	W =  90.000 deg,	P =   0.000 deg,	R =   90.000 deg
};
P[1529]{
   GP1:
	UF : 0, UT : 6,		CONFIG : 'N U T, 0, 0, 0',
	X =  489.358  mm,	Y =   -298.597  mm,	Z =   -262.804  mm,
	W =  90.000 deg,	P =   0.000 deg,	R =   90.000 deg
};
P[1530]{
   GP1:
	UF : 0, UT : 6,		CONFIG : 'N U T, 0, 0, 0',
	X =  488.486  mm,	Y =   -297.265  mm,	Z =   -263.052  mm,
	W =  90.000 deg,	P =   0.000 deg,	R =   90.000 deg
};
P[1531]{
   GP1:
	UF : 0, UT : 6,		CONFIG : 'N U T, 0, 0, 0',
	X =  487.911  mm,	Y =   -296.359  mm,	Z =   -263.179  mm,
	W =  90.000 deg,	P =   0.000 deg,	R =   90.000 deg
};
P[1532]{
   GP1:
	UF : 0, UT : 6,		CONFIG : 'N U T, 0, 0, 0',
	X =  487.436  mm,	Y =   -295.414  mm,	Z =   -263.006  mm,
	W =  90.000 deg,	P =   0.000 deg,	R =   90.000 deg
};
P[1533]{
   GP1:
	UF : 0, UT : 6,		CONFIG : 'N U T, 0, 0, 0',
	X =  485.822  mm,	Y =   -292.714  mm,	Z =   -263.142  mm,
	W =  90.000 deg,	P =   0.000 deg,	R =   90.000 deg
};
P[1534]{
   GP1:
	UF : 0, UT : 6,		CONFIG : 'N U T, 0, 0, 0',
	X =  485.360  mm,	Y =   -291.792  mm,	Z =   -262.970  mm,
	W =  90.000 deg,	P =   0.000 deg,	R =   90.000 deg
};
P[1535]{
   GP1:
	UF : 0, UT : 6,		CONFIG : 'N U T, 0, 0, 0',
	X =  484.532  mm,	Y =   -290.400  mm,	Z =   -263.029  mm,
	W =  90.000 deg,	P =   0.000 deg,	R =   90.000 deg
};
P[1536]{
   GP1:
	UF : 0, UT : 6,		CONFIG : 'N U T, 0, 0, 0',
	X =  483.396  mm,	Y =   -288.373  mm,	Z =   -262.945  mm,
	W =  90.000 deg,	P =   0.000 deg,	R =   90.000 deg
};
P[1537]{
   GP1:
	UF : 0, UT : 6,		CONFIG : 'N U T, 0, 0, 0',
	X =  482.953  mm,	Y =   -287.646  mm,	Z =   -263.001  mm,
	W =  90.000 deg,	P =   0.000 deg,	R =   90.000 deg
};
P[1538]{
   GP1:
	UF : 0, UT : 6,		CONFIG : 'N U T, 0, 0, 0',
	X =  482.093  mm,	Y =   -286.165  mm,	Z =   -263.010  mm,
	W =  90.000 deg,	P =   0.000 deg,	R =   90.000 deg
};
P[1539]{
   GP1:
	UF : 0, UT : 6,		CONFIG : 'N U T, 0, 0, 0',
	X =  480.613  mm,	Y =   -283.699  mm,	Z =   -263.148  mm,
	W =  90.000 deg,	P =   0.000 deg,	R =   90.000 deg
};
P[1540]{
   GP1:
	UF : 0, UT : 6,		CONFIG : 'N U T, 0, 0, 0',
	X =  479.567  mm,	Y =   -281.920  mm,	Z =   -263.196  mm,
	W =  90.000 deg,	P =   0.000 deg,	R =   90.000 deg
};
P[1541]{
   GP1:
	UF : 0, UT : 6,		CONFIG : 'N U T, 0, 0, 0',
	X =  478.631  mm,	Y =   -280.161  mm,	Z =   -263.002  mm,
	W =  90.000 deg,	P =   0.000 deg,	R =   90.000 deg
};
P[1542]{
   GP1:
	UF : 0, UT : 6,		CONFIG : 'N U T, 0, 0, 0',
	X =  478.100  mm,	Y =   -279.216  mm,	Z =   -262.965  mm,
	W =  90.000 deg,	P =   0.000 deg,	R =   90.000 deg
};
P[1543]{
   GP1:
	UF : 0, UT : 6,		CONFIG : 'N U T, 0, 0, 0',
	X =  477.160  mm,	Y =   -277.535  mm,	Z =   -262.892  mm,
	W =  90.000 deg,	P =   0.000 deg,	R =   90.000 deg
};
P[1544]{
   GP1:
	UF : 0, UT : 6,		CONFIG : 'N U T, 0, 0, 0',
	X =  476.282  mm,	Y =   -276.005  mm,	Z =   -262.880  mm,
	W =  90.000 deg,	P =   0.000 deg,	R =   90.000 deg
};
P[1545]{
   GP1:
	UF : 0, UT : 6,		CONFIG : 'N U T, 0, 0, 0',
	X =  475.643  mm,	Y =   -275.130  mm,	Z =   -263.205  mm,
	W =  90.000 deg,	P =   0.000 deg,	R =   90.000 deg
};
P[1546]{
   GP1:
	UF : 0, UT : 6,		CONFIG : 'N U T, 0, 0, 0',
	X =  473.837  mm,	Y =   -272.025  mm,	Z =   -263.237  mm,
	W =  90.000 deg,	P =   0.000 deg,	R =   90.000 deg
};
P[1547]{
   GP1:
	UF : 0, UT : 6,		CONFIG : 'N U T, 0, 0, 0',
	X =  472.547  mm,	Y =   -269.731  mm,	Z =   -263.150  mm,
	W =  90.000 deg,	P =   0.000 deg,	R =   90.000 deg
};
P[1548]{
   GP1:
	UF : 0, UT : 6,		CONFIG : 'N U T, 0, 0, 0',
	X =  471.867  mm,	Y =   -268.518  mm,	Z =   -263.103  mm,
	W =  90.000 deg,	P =   0.000 deg,	R =   90.000 deg
};
P[1549]{
   GP1:
	UF : 0, UT : 6,		CONFIG : 'N U T, 0, 0, 0',
	X =  470.788  mm,	Y =   -266.711  mm,	Z =   -263.187  mm,
	W =  90.000 deg,	P =   0.000 deg,	R =   90.000 deg
};
P[1550]{
   GP1:
	UF : 0, UT : 6,		CONFIG : 'N U T, 0, 0, 0',
	X =  469.454  mm,	Y =   -264.407  mm,	Z =   -263.197  mm,
	W =  90.000 deg,	P =   0.000 deg,	R =   90.000 deg
};
P[1551]{
   GP1:
	UF : 0, UT : 6,		CONFIG : 'N U T, 0, 0, 0',
	X =  468.882  mm,	Y =   -263.356  mm,	Z =   -263.113  mm,
	W =  90.000 deg,	P =   0.000 deg,	R =   90.000 deg
};
P[1552]{
   GP1:
	UF : 0, UT : 6,		CONFIG : 'N U T, 0, 0, 0',
	X =  468.477  mm,	Y =   -262.544  mm,	Z =   -262.960  mm,
	W =  90.000 deg,	P =   0.000 deg,	R =   90.000 deg
};
P[1553]{
   GP1:
	UF : 0, UT : 6,		CONFIG : 'N U T, 0, 0, 0',
	X =  467.176  mm,	Y =   -260.442  mm,	Z =   -263.171  mm,
	W =  90.000 deg,	P =   0.000 deg,	R =   90.000 deg
};
P[1554]{
   GP1:
	UF : 0, UT : 6,		CONFIG : 'N U T, 0, 0, 0',
	X =  466.411  mm,	Y =   -259.155  mm,	Z =   -263.222  mm,
	W =  90.000 deg,	P =   0.000 deg,	R =   90.000 deg
};
P[1555]{
   GP1:
	UF : 0, UT : 6,		CONFIG : 'N U T, 0, 0, 0',
	X =  465.241  mm,	Y =   -256.952  mm,	Z =   -262.976  mm,
	W =  90.000 deg,	P =   0.000 deg,	R =   90.000 deg
};
P[1556]{
   GP1:
	UF : 0, UT : 6,		CONFIG : 'N U T, 0, 0, 0',
	X =  464.232  mm,	Y =   -255.232  mm,	Z =   -263.015  mm,
	W =  90.000 deg,	P =   0.000 deg,	R =   90.000 deg
};
P[1557]{
   GP1:
	UF : 0, UT : 6,		CONFIG : 'N U T, 0, 0, 0',
	X =  463.784  mm,	Y =   -254.434  mm,	Z =   -262.984  mm,
	W =  90.000 deg,	P =   0.000 deg,	R =   90.000 deg
};
P[1558]{
   GP1:
	UF : 0, UT : 6,		CONFIG : 'N U T, 0, 0, 0',
	X =  462.902  mm,	Y =   -253.033  mm,	Z =   -263.160  mm,
	W =  90.000 deg,	P =   0.000 deg,	R =   90.000 deg
};
P[1559]{
   GP1:
	UF : 0, UT : 6,		CONFIG : 'N U T, 0, 0, 0',
	X =  462.571  mm,	Y =   -252.324  mm,	Z =   -262.969  mm,
	W =  90.000 deg,	P =   0.000 deg,	R =   90.000 deg
};
P[1560]{
   GP1:
	UF : 0, UT : 6,		CONFIG : 'N U T, 0, 0, 0',
	X =  460.908  mm,	Y =   -249.546  mm,	Z =   -263.113  mm,
	W =  90.000 deg,	P =   0.000 deg,	R =   90.000 deg
};
P[1561]{
   GP1:
	UF : 0, UT : 6,		CONFIG : 'N U T, 0, 0, 0',
	X =  459.581  mm,	Y =   -247.266  mm,	Z =   -263.139  mm,
	W =  90.000 deg,	P =   0.000 deg,	R =   90.000 deg
};
P[1562]{
   GP1:
	UF : 0, UT : 6,		CONFIG : 'N U T, 0, 0, 0',
	X =  458.765  mm,	Y =   -245.901  mm,	Z =   -263.206  mm,
	W =  90.000 deg,	P =   0.000 deg,	R =   90.000 deg
};
P[1563]{
   GP1:
	UF : 0, UT : 6,		CONFIG : 'N U T, 0, 0, 0',
	X =  457.689  mm,	Y =   -243.918  mm,	Z =   -263.039  mm,
	W =  90.000 deg,	P =   0.000 deg,	R =   90.000 deg
};
P[1564]{
   GP1:
	UF : 0, UT : 6,		CONFIG : 'N U T, 0, 0, 0',
	X =  456.741  mm,	Y =   -242.187  mm,	Z =   -262.917  mm,
	W =  90.000 deg,	P =   0.000 deg,	R =   90.000 deg
};
P[1565]{
   GP1:
	UF : 0, UT : 6,		CONFIG : 'N U T, 0, 0, 0',
	X =  456.319  mm,	Y =   -241.589  mm,	Z =   -263.103  mm,
	W =  90.000 deg,	P =   0.000 deg,	R =   90.000 deg
};
P[1566]{
   GP1:
	UF : 0, UT : 6,		CONFIG : 'N U T, 0, 0, 0',
	X =  455.661  mm,	Y =   -240.265  mm,	Z =   -262.842  mm,
	W =  90.000 deg,	P =   0.000 deg,	R =   90.000 deg
};
P[1567]{
   GP1:
	UF : 0, UT : 6,		CONFIG : 'N U T, 0, 0, 0',
	X =  454.825  mm,	Y =   -238.885  mm,	Z =   -262.936  mm,
	W =  90.000 deg,	P =   0.000 deg,	R =   90.000 deg
};
P[1568]{
   GP1:
	UF : 0, UT : 6,		CONFIG : 'N U T, 0, 0, 0',
	X =  452.965  mm,	Y =   -235.714  mm,	Z =   -263.009  mm,
	W =  90.000 deg,	P =   0.000 deg,	R =   90.000 deg
};
P[1569]{
   GP1:
	UF : 0, UT : 6,		CONFIG : 'N U T, 0, 0, 0',
	X =  452.402  mm,	Y =   -234.770  mm,	Z =   -263.054  mm,
	W =  90.000 deg,	P =   0.000 deg,	R =   90.000 deg
};
P[1570]{
   GP1:
	UF : 0, UT : 6,		CONFIG : 'N U T, 0, 0, 0',
	X =  451.666  mm,	Y =   -233.332  mm,	Z =   -262.824  mm,
	W =  90.000 deg,	P =   0.000 deg,	R =   90.000 deg
};
P[1571]{
   GP1:
	UF : 0, UT : 6,		CONFIG : 'N U T, 0, 0, 0',
	X =  449.809  mm,	Y =   -230.157  mm,	Z =   -262.879  mm,
	W =  90.000 deg,	P =   0.000 deg,	R =   90.000 deg
};
P[1572]{
   GP1:
	UF : 0, UT : 6,		CONFIG : 'N U T, 0, 0, 0',
	X =  448.786  mm,	Y =   -228.608  mm,	Z =   -263.191  mm,
	W =  90.000 deg,	P =   0.000 deg,	R =   90.000 deg
};
P[1573]{
   GP1:
	UF : 0, UT : 6,		CONFIG : 'N U T, 0, 0, 0',
	X =  446.779  mm,	Y =   -225.065  mm,	Z =   -263.099  mm,
	W =  90.000 deg,	P =   0.000 deg,	R =   90.000 deg
};
P[1574]{
   GP1:
	UF : 0, UT : 6,		CONFIG : 'N U T, 0, 0, 0',
	X =  445.861  mm,	Y =   -223.520  mm,	Z =   -263.160  mm,
	W =  90.000 deg,	P =   0.000 deg,	R =   90.000 deg
};
P[1575]{
   GP1:
	UF : 0, UT : 6,		CONFIG : 'N U T, 0, 0, 0',
	X =  444.870  mm,	Y =   -221.679  mm,	Z =   -262.988  mm,
	W =  90.000 deg,	P =   0.000 deg,	R =   90.000 deg
};
P[1576]{
   GP1:
	UF : 0, UT : 6,		CONFIG : 'N U T, 0, 0, 0',
	X =  444.103  mm,	Y =   -220.377  mm,	Z =   -263.023  mm,
	W =  90.000 deg,	P =   0.000 deg,	R =   90.000 deg
};
P[1577]{
   GP1:
	UF : 0, UT : 6,		CONFIG : 'N U T, 0, 0, 0',
	X =  442.799  mm,	Y =   -218.282  mm,	Z =   -263.252  mm,
	W =  90.000 deg,	P =   0.000 deg,	R =   90.000 deg
};
P[1578]{
   GP1:
	UF : 0, UT : 6,		CONFIG : 'N U T, 0, 0, 0',
	X =  441.471  mm,	Y =   -215.902  mm,	Z =   -263.142  mm,
	W =  90.000 deg,	P =   0.000 deg,	R =   90.000 deg
};
P[1579]{
   GP1:
	UF : 0, UT : 6,		CONFIG : 'N U T, 0, 0, 0',
	X =  439.128  mm,	Y =   -211.770  mm,	Z =   -263.038  mm,
	W =  90.000 deg,	P =   0.000 deg,	R =   90.000 deg
};
P[1580]{
   GP1:
	UF : 0, UT : 6,		CONFIG : 'N U T, 0, 0, 0',
	X =  438.540  mm,	Y =   -210.657  mm,	Z =   -262.904  mm,
	W =  90.000 deg,	P =   0.000 deg,	R =   90.000 deg
};
P[1581]{
   GP1:
	UF : 0, UT : 6,		CONFIG : 'N U T, 0, 0, 0',
	X =  437.892  mm,	Y =   -209.754  mm,	Z =   -263.213  mm,
	W =  90.000 deg,	P =   0.000 deg,	R =   90.000 deg
};
P[1582]{
   GP1:
	UF : 0, UT : 6,		CONFIG : 'N U T, 0, 0, 0',
	X =  437.474  mm,	Y =   -208.890  mm,	Z =   -263.015  mm,
	W =  90.000 deg,	P =   0.000 deg,	R =   90.000 deg
};
P[1583]{
   GP1:
	UF : 0, UT : 6,		CONFIG : 'N U T, 0, 0, 0',
	X =  436.948  mm,	Y =   -207.939  mm,	Z =   -262.959  mm,
	W =  90.000 deg,	P =   0.000 deg,	R =   90.000 deg
};
P[1584]{
   GP1:
	UF : 0, UT : 6,		CONFIG : 'N U T, 0, 0, 0',
	X =  435.779  mm,	Y =   -205.907  mm,	Z =   -262.948  mm,
	W =  90.000 deg,	P =   0.000 deg,	R =   90.000 deg
};
P[1585]{
   GP1:
	UF : 0, UT : 6,		CONFIG : 'N U T, 0, 0, 0',
	X =  434.758  mm,	Y =   -204.064  mm,	Z =   -262.845  mm,
	W =  90.000 deg,	P =   0.000 deg,	R =   90.000 deg
};
P[1586]{
   GP1:
	UF : 0, UT : 6,		CONFIG : 'N U T, 0, 0, 0',
	X =  433.658  mm,	Y =   -202.324  mm,	Z =   -263.077  mm,
	W =  90.000 deg,	P =   0.000 deg,	R =   90.000 deg
};
P[1587]{
   GP1:
	UF : 0, UT : 6,		CONFIG : 'N U T, 0, 0, 0',
	X =  432.346  mm,	Y =   -199.899  mm,	Z =   -262.861  mm,
	W =  90.000 deg,	P =   0.000 deg,	R =   90.000 deg
};
P[1588]{
   GP1:
	UF : 0, UT : 6,		CONFIG : 'N U T, 0, 0, 0',
	X =  431.514  mm,	Y =   -198.665  mm,	Z =   -263.152  mm,
	W =  90.000 deg,	P =   0.000 deg,	R =   90.000 deg
};
P[1589]{
   GP1:
	UF : 0, UT : 6,		CONFIG : 'N U T, 0, 0, 0',
	X =  429.834  mm,	Y =   -195.647  mm,	Z =   -263.001  mm,
	W =  90.000 deg,	P =   0.000 deg,	R =   90.000 deg
};
P[1590]{
   GP1:
	UF : 0, UT : 6,		CONFIG : 'N U T, 0, 0, 0',
	X =  426.599  mm,	Y =   -190.074  mm,	Z =   -263.043  mm,
	W =  90.000 deg,	P =   0.000 deg,	R =   90.000 deg
};
P[1591]{
   GP1:
	UF : 0, UT : 6,		CONFIG : 'N U T, 0, 0, 0',
	X =  425.932  mm,	Y =   -188.910  mm,	Z =   -263.028  mm,
	W =  90.000 deg,	P =   0.000 deg,	R =   90.000 deg
};
P[1592]{
   GP1:
	UF : 0, UT : 6,		CONFIG : 'N U T, 0, 0, 0',
	X =  425.483  mm,	Y =   -187.966  mm,	Z =   -262.797  mm,
	W =  90.000 deg,	P =   0.000 deg,	R =   90.000 deg
};
P[1593]{
   GP1:
	UF : 0, UT : 6,		CONFIG : 'N U T, 0, 0, 0',
	X =  425.046  mm,	Y =   -187.431  mm,	Z =   -263.109  mm,
	W =  90.000 deg,	P =   0.000 deg,	R =   90.000 deg
};
P[1594]{
   GP1:
	UF : 0, UT : 6,		CONFIG : 'N U T, 0, 0, 0',
	X =  424.035  mm,	Y =   -185.506  mm,	Z =   -262.865  mm,
	W =  90.000 deg,	P =   0.000 deg,	R =   90.000 deg
};
P[1595]{
   GP1:
	UF : 0, UT : 6,		CONFIG : 'N U T, 0, 0, 0',
	X =  423.248  mm,	Y =   -184.271  mm,	Z =   -263.042  mm,
	W =  90.000 deg,	P =   0.000 deg,	R =   90.000 deg
};
P[1596]{
   GP1:
	UF : 0, UT : 6,		CONFIG : 'N U T, 0, 0, 0',
	X =  422.871  mm,	Y =   -183.702  mm,	Z =   -263.158  mm,
	W =  90.000 deg,	P =   0.000 deg,	R =   90.000 deg
};
P[1597]{
   GP1:
	UF : 0, UT : 6,		CONFIG : 'N U T, 0, 0, 0',
	X =  422.029  mm,	Y =   -182.194  mm,	Z =   -263.092  mm,
	W =  90.000 deg,	P =   0.000 deg,	R =   90.000 deg
};
P[1598]{
   GP1:
	UF : 0, UT : 6,		CONFIG : 'N U T, 0, 0, 0',
	X =  421.712  mm,	Y =   -181.429  mm,	Z =   -262.788  mm,
	W =  90.000 deg,	P =   0.000 deg,	R =   90.000 deg
};
P[1599]{
   GP1:
	UF : 0, UT : 6,		CONFIG : 'N U T, 0, 0, 0',
	X =  420.760  mm,	Y =   -179.893  mm,	Z =   -262.947  mm,
	W =  90.000 deg,	P =   0.000 deg,	R =   90.000 deg
};
P[1600]{
   GP1:
	UF : 0, UT : 6,		CONFIG : 'N U T, 0, 0, 0',
	X =  418.495  mm,	Y =   -176.142  mm,	Z =   -263.188  mm,
	W =  90.000 deg,	P =   0.000 deg,	R =   90.000 deg
};
P[1601]{
   GP1:
	UF : 0, UT : 6,		CONFIG : 'N U T, 0, 0, 0',
	X =  416.729  mm,	Y =   -173.099  mm,	Z =   -263.209  mm,
	W =  90.000 deg,	P =   0.000 deg,	R =   90.000 deg
};
P[1602]{
   GP1:
	UF : 0, UT : 6,		CONFIG : 'N U T, 0, 0, 0',
	X =  416.215  mm,	Y =   -172.155  mm,	Z =   -263.132  mm,
	W =  90.000 deg,	P =   0.000 deg,	R =   90.000 deg
};
P[1603]{
   GP1:
	UF : 0, UT : 6,		CONFIG : 'N U T, 0, 0, 0',
	X =  415.460  mm,	Y =   -170.608  mm,	Z =   -262.798  mm,
	W =  90.000 deg,	P =   0.000 deg,	R =   90.000 deg
};
P[1604]{
   GP1:
	UF : 0, UT : 6,		CONFIG : 'N U T, 0, 0, 0',
	X =  414.951  mm,	Y =   -170.002  mm,	Z =   -263.184  mm,
	W =  90.000 deg,	P =   0.000 deg,	R =   90.000 deg
};
P[1605]{
   GP1:
	UF : 0, UT : 6,		CONFIG : 'N U T, 0, 0, 0',
	X =  413.920  mm,	Y =   -168.065  mm,	Z =   -262.973  mm,
	W =  90.000 deg,	P =   0.000 deg,	R =   90.000 deg
};
P[1606]{
   GP1:
	UF : 0, UT : 6,		CONFIG : 'N U T, 0, 0, 0',
	X =  412.944  mm,	Y =   -166.529  mm,	Z =   -263.191  mm,
	W =  90.000 deg,	P =   0.000 deg,	R =   90.000 deg
};
P[1607]{
   GP1:
	UF : 0, UT : 6,		CONFIG : 'N U T, 0, 0, 0',
	X =  411.430  mm,	Y =   -163.848  mm,	Z =   -263.106  mm,
	W =  90.000 deg,	P =   0.000 deg,	R =   90.000 deg
};
P[1608]{
   GP1:
	UF : 0, UT : 6,		CONFIG : 'N U T, 0, 0, 0',
	X =  411.083  mm,	Y =   -163.130  mm,	Z =   -262.940  mm,
	W =  90.000 deg,	P =   0.000 deg,	R =   90.000 deg
};
P[1609]{
   GP1:
	UF : 0, UT : 6,		CONFIG : 'N U T, 0, 0, 0',
	X =  410.279  mm,	Y =   -161.767  mm,	Z =   -262.982  mm,
	W =  90.000 deg,	P =   0.000 deg,	R =   90.000 deg
};
P[1610]{
   GP1:
	UF : 0, UT : 6,		CONFIG : 'N U T, 0, 0, 0',
	X =  409.631  mm,	Y =   -160.731  mm,	Z =   -263.102  mm,
	W =  90.000 deg,	P =   0.000 deg,	R =   90.000 deg
};
P[1611]{
   GP1:
	UF : 0, UT : 6,		CONFIG : 'N U T, 0, 0, 0',
	X =  407.922  mm,	Y =   -157.760  mm,	Z =   -263.088  mm,
	W =  90.000 deg,	P =   0.000 deg,	R =   90.000 deg
};
P[1612]{
   GP1:
	UF : 0, UT : 6,		CONFIG : 'N U T, 0, 0, 0',
	X =  406.251  mm,	Y =   -154.891  mm,	Z =   -263.124  mm,
	W =  90.000 deg,	P =   0.000 deg,	R =   90.000 deg
};
P[1613]{
   GP1:
	UF : 0, UT : 6,		CONFIG : 'N U T, 0, 0, 0',
	X =  403.461  mm,	Y =   -149.918  mm,	Z =   -262.925  mm,
	W =  90.000 deg,	P =   0.000 deg,	R =   90.000 deg
};
P[1614]{
   GP1:
	UF : 0, UT : 6,		CONFIG : 'N U T, 0, 0, 0',
	X =  402.068  mm,	Y =   -147.568  mm,	Z =   -263.014  mm,
	W =  90.000 deg,	P =   0.000 deg,	R =   90.000 deg
};
P[1615]{
   GP1:
	UF : 0, UT : 6,		CONFIG : 'N U T, 0, 0, 0',
	X =  401.082  mm,	Y =   -145.926  mm,	Z =   -263.105  mm,
	W =  90.000 deg,	P =   0.000 deg,	R =   90.000 deg
};
P[1616]{
   GP1:
	UF : 0, UT : 6,		CONFIG : 'N U T, 0, 0, 0',
	X =  400.512  mm,	Y =   -144.717  mm,	Z =   -262.796  mm,
	W =  90.000 deg,	P =   0.000 deg,	R =   90.000 deg
};
P[1617]{
   GP1:
	UF : 0, UT : 6,		CONFIG : 'N U T, 0, 0, 0',
	X =  400.093  mm,	Y =   -144.000  mm,	Z =   -262.806  mm,
	W =  90.000 deg,	P =   0.000 deg,	R =   90.000 deg
};
P[1618]{
   GP1:
	UF : 0, UT : 6,		CONFIG : 'N U T, 0, 0, 0',
	X =  398.900  mm,	Y =   -142.145  mm,	Z =   -263.103  mm,
	W =  90.000 deg,	P =   0.000 deg,	R =   90.000 deg
};
P[1619]{
   GP1:
	UF : 0, UT : 6,		CONFIG : 'N U T, 0, 0, 0',
	X =  397.403  mm,	Y =   -139.331  mm,	Z =   -262.792  mm,
	W =  90.000 deg,	P =   0.000 deg,	R =   90.000 deg
};
P[1620]{
   GP1:
	UF : 0, UT : 6,		CONFIG : 'N U T, 0, 0, 0',
	X =  396.568  mm,	Y =   -138.118  mm,	Z =   -263.120  mm,
	W =  90.000 deg,	P =   0.000 deg,	R =   90.000 deg
};
P[1621]{
   GP1:
	UF : 0, UT : 6,		CONFIG : 'N U T, 0, 0, 0',
	X =  396.064  mm,	Y =   -137.155  mm,	Z =   -262.994  mm,
	W =  90.000 deg,	P =   0.000 deg,	R =   90.000 deg
};
P[1622]{
   GP1:
	UF : 0, UT : 6,		CONFIG : 'N U T, 0, 0, 0',
	X =  395.600  mm,	Y =   -136.355  mm,	Z =   -262.998  mm,
	W =  90.000 deg,	P =   0.000 deg,	R =   90.000 deg
};
P[1623]{
   GP1:
	UF : 0, UT : 6,		CONFIG : 'N U T, 0, 0, 0',
	X =  393.626  mm,	Y =   -133.094  mm,	Z =   -263.218  mm,
	W =  90.000 deg,	P =   0.000 deg,	R =   90.000 deg
};
P[1624]{
   GP1:
	UF : 0, UT : 6,		CONFIG : 'N U T, 0, 0, 0',
	X =  392.762  mm,	Y =   -131.420  mm,	Z =   -262.969  mm,
	W =  90.000 deg,	P =   0.000 deg,	R =   90.000 deg
};
P[1625]{
   GP1:
	UF : 0, UT : 6,		CONFIG : 'N U T, 0, 0, 0',
	X =  391.901  mm,	Y =   -129.970  mm,	Z =   -263.028  mm,
	W =  90.000 deg,	P =   0.000 deg,	R =   90.000 deg
};
P[1626]{
   GP1:
	UF : 0, UT : 6,		CONFIG : 'N U T, 0, 0, 0',
	X =  391.473  mm,	Y =   -129.173  mm,	Z =   -262.952  mm,
	W =  90.000 deg,	P =   0.000 deg,	R =   90.000 deg
};
P[1627]{
   GP1:
	UF : 0, UT : 6,		CONFIG : 'N U T, 0, 0, 0',
	X =  390.645  mm,	Y =   -127.611  mm,	Z =   -262.770  mm,
	W =  90.000 deg,	P =   0.000 deg,	R =   90.000 deg
};
P[1628]{
   GP1:
	UF : 0, UT : 6,		CONFIG : 'N U T, 0, 0, 0',
	X =  390.141  mm,	Y =   -127.012  mm,	Z =   -263.154  mm,
	W =  90.000 deg,	P =   0.000 deg,	R =   90.000 deg
};
P[1629]{
   GP1:
	UF : 0, UT : 6,		CONFIG : 'N U T, 0, 0, 0',
	X =  389.441  mm,	Y =   -125.590  mm,	Z =   -262.861  mm,
	W =  90.000 deg,	P =   0.000 deg,	R =   90.000 deg
};
P[1630]{
   GP1:
	UF : 0, UT : 6,		CONFIG : 'N U T, 0, 0, 0',
	X =  387.124  mm,	Y =   -121.753  mm,	Z =   -263.107  mm,
	W =  90.000 deg,	P =   0.000 deg,	R =   90.000 deg
};
P[1631]{
   GP1:
	UF : 0, UT : 6,		CONFIG : 'N U T, 0, 0, 0',
	X =  386.314  mm,	Y =   -120.317  mm,	Z =   -263.062  mm,
	W =  90.000 deg,	P =   0.000 deg,	R =   90.000 deg
};
P[1632]{
   GP1:
	UF : 0, UT : 6,		CONFIG : 'N U T, 0, 0, 0',
	X =  385.225  mm,	Y =   -118.429  mm,	Z =   -263.057  mm,
	W =  90.000 deg,	P =   0.000 deg,	R =   90.000 deg
};
P[1633]{
   GP1:
	UF : 0, UT : 6,		CONFIG : 'N U T, 0, 0, 0',
	X =  384.441  mm,	Y =   -116.898  mm,	Z =   -262.814  mm,
	W =  90.000 deg,	P =   0.000 deg,	R =   90.000 deg
};
P[1634]{
   GP1:
	UF : 0, UT : 6,		CONFIG : 'N U T, 0, 0, 0',
	X =  382.319  mm,	Y =   -113.417  mm,	Z =   -263.088  mm,
	W =  90.000 deg,	P =   0.000 deg,	R =   90.000 deg
};
P[1635]{
   GP1:
	UF : 0, UT : 6,		CONFIG : 'N U T, 0, 0, 0',
	X =  381.654  mm,	Y =   -112.274  mm,	Z =   -263.100  mm,
	W =  90.000 deg,	P =   0.000 deg,	R =   90.000 deg
};
P[1636]{
   GP1:
	UF : 0, UT : 6,		CONFIG : 'N U T, 0, 0, 0',
	X =  380.710  mm,	Y =   -110.408  mm,	Z =   -262.778  mm,
	W =  90.000 deg,	P =   0.000 deg,	R =   90.000 deg
};
P[1637]{
   GP1:
	UF : 0, UT : 6,		CONFIG : 'N U T, 0, 0, 0',
	X =  379.963  mm,	Y =   -109.240  mm,	Z =   -262.951  mm,
	W =  90.000 deg,	P =   0.000 deg,	R =   90.000 deg
};
P[1638]{
   GP1:
	UF : 0, UT : 6,		CONFIG : 'N U T, 0, 0, 0',
	X =  377.252  mm,	Y =   -104.569  mm,	Z =   -262.988  mm,
	W =  90.000 deg,	P =   0.000 deg,	R =   90.000 deg
};
P[1639]{
   GP1:
	UF : 0, UT : 6,		CONFIG : 'N U T, 0, 0, 0',
	X =  375.992  mm,	Y =   -102.293  mm,	Z =   -262.856  mm,
	W =  90.000 deg,	P =   0.000 deg,	R =   90.000 deg
};
P[1640]{
   GP1:
	UF : 0, UT : 6,		CONFIG : 'N U T, 0, 0, 0',
	X =  374.863  mm,	Y =   -100.498  mm,	Z =   -263.080  mm,
	W =  90.000 deg,	P =   0.000 deg,	R =   90.000 deg
};
P[1641]{
   GP1:
	UF : 0, UT : 6,		CONFIG : 'N U T, 0, 0, 0',
	X =  374.474  mm,	Y =   -99.912  mm,	Z =   -263.205  mm,
	W =  90.000 deg,	P =   0.000 deg,	R =   90.000 deg
};
P[1642]{
   GP1:
	UF : 0, UT : 6,		CONFIG : 'N U T, 0, 0, 0',
	X =  373.888  mm,	Y =   -98.873  mm,	Z =   -263.168  mm,
	W =  90.000 deg,	P =   0.000 deg,	R =   90.000 deg
};
P[1643]{
   GP1:
	UF : 0, UT : 6,		CONFIG : 'N U T, 0, 0, 0',
	X =  373.663  mm,	Y =   -98.250  mm,	Z =   -262.841  mm,
	W =  90.000 deg,	P =   0.000 deg,	R =   90.000 deg
};
P[1644]{
   GP1:
	UF : 0, UT : 6,		CONFIG : 'N U T, 0, 0, 0',
	X =  372.355  mm,	Y =   -96.276  mm,	Z =   -263.250  mm,
	W =  90.000 deg,	P =   0.000 deg,	R =   90.000 deg
};
P[1645]{
   GP1:
	UF : 0, UT : 6,		CONFIG : 'N U T, 0, 0, 0',
	X =  372.087  mm,	Y =   -95.536  mm,	Z =   -262.863  mm,
	W =  90.000 deg,	P =   0.000 deg,	R =   90.000 deg
};
P[1646]{
   GP1:
	UF : 0, UT : 6,		CONFIG : 'N U T, 0, 0, 0',
	X =  370.787  mm,	Y =   -93.521  mm,	Z =   -263.196  mm,
	W =  90.000 deg,	P =   0.000 deg,	R =   90.000 deg
};
P[1647]{
   GP1:
	UF : 0, UT : 6,		CONFIG : 'N U T, 0, 0, 0',
	X =  370.163  mm,	Y =   -92.365  mm,	Z =   -263.088  mm,
	W =  90.000 deg,	P =   0.000 deg,	R =   90.000 deg
};
P[1648]{
   GP1:
	UF : 0, UT : 6,		CONFIG : 'N U T, 0, 0, 0',
	X =  369.057  mm,	Y =   -90.533  mm,	Z =   -263.207  mm,
	W =  90.000 deg,	P =   0.000 deg,	R =   90.000 deg
};
P[1649]{
   GP1:
	UF : 0, UT : 6,		CONFIG : 'N U T, 0, 0, 0',
	X =  367.390  mm,	Y =   -87.837  mm,	Z =   -263.021  mm,
	W =  90.000 deg,	P =   0.000 deg,	R =   90.000 deg
};
P[1650]{
   GP1:
	UF : 0, UT : 6,		CONFIG : 'N U T, 0, 0, 0',
	X =  366.347  mm,	Y =   -86.500  mm,	Z =   -263.021  mm,
	W =  90.000 deg,	P =   0.000 deg,	R =   90.000 deg
};
P[1651]{
   GP1:
	UF : 0, UT : 6,		CONFIG : 'N U T, 0, 0, 0',
	X =  365.186  mm,	Y =   -85.520  mm,	Z =   -263.165  mm,
	W =  90.000 deg,	P =   0.000 deg,	R =   90.000 deg
};
P[1652]{
   GP1:
	UF : 0, UT : 6,		CONFIG : 'N U T, 0, 0, 0',
	X =  363.058  mm,	Y =   -84.038  mm,	Z =   -263.228  mm,
	W =  90.000 deg,	P =   0.000 deg,	R =   90.000 deg
};
P[1653]{
   GP1:
	UF : 0, UT : 6,		CONFIG : 'N U T, 0, 0, 0',
	X =  362.412  mm,	Y =   -83.671  mm,	Z =   -263.193  mm,
	W =  90.000 deg,	P =   0.000 deg,	R =   90.000 deg
};
P[1654]{
   GP1:
	UF : 0, UT : 6,		CONFIG : 'N U T, 0, 0, 0',
	X =  361.565  mm,	Y =   -83.157  mm,	Z =   -263.036  mm,
	W =  90.000 deg,	P =   0.000 deg,	R =   90.000 deg
};
P[1655]{
   GP1:
	UF : 0, UT : 6,		CONFIG : 'N U T, 0, 0, 0',
	X =  357.539  mm,	Y =   -82.314  mm,	Z =   -263.191  mm,
	W =  90.000 deg,	P =   0.000 deg,	R =   90.000 deg
};
P[1656]{
   GP1:
	UF : 0, UT : 6,		CONFIG : 'N U T, 0, 0, 0',
	X =  356.612  mm,	Y =   -82.227  mm,	Z =   -263.068  mm,
	W =  90.000 deg,	P =   0.000 deg,	R =   90.000 deg
};
P[1657]{
   GP1:
	UF : 0, UT : 6,		CONFIG : 'N U T, 0, 0, 0',
	X =  355.608  mm,	Y =   -82.192  mm,	Z =   -262.999  mm,
	W =  90.000 deg,	P =   0.000 deg,	R =   90.000 deg
};
P[1658]{
   GP1:
	UF : 0, UT : 6,		CONFIG : 'N U T, 0, 0, 0',
	X =  354.673  mm,	Y =   -82.287  mm,	Z =   -262.946  mm,
	W =  90.000 deg,	P =   0.000 deg,	R =   90.000 deg
};
P[1659]{
   GP1:
	UF : 0, UT : 6,		CONFIG : 'N U T, 0, 0, 0',
	X =  353.716  mm,	Y =   -82.545  mm,	Z =   -263.088  mm,
	W =  90.000 deg,	P =   0.000 deg,	R =   90.000 deg
};
P[1660]{
   GP1:
	UF : 0, UT : 6,		CONFIG : 'N U T, 0, 0, 0',
	X =  350.442  mm,	Y =   -83.670  mm,	Z =   -263.077  mm,
	W =  90.000 deg,	P =   0.000 deg,	R =   90.000 deg
};
P[1661]{
   GP1:
	UF : 0, UT : 6,		CONFIG : 'N U T, 0, 0, 0',
	X =  347.275  mm,	Y =   -85.379  mm,	Z =   -263.080  mm,
	W =  90.000 deg,	P =   0.000 deg,	R =   90.000 deg
};
P[1662]{
   GP1:
	UF : 0, UT : 6,		CONFIG : 'N U T, 0, 0, 0',
	X =  345.761  mm,	Y =   -86.280  mm,	Z =   -263.144  mm,
	W =  90.000 deg,	P =   0.000 deg,	R =   90.000 deg
};
P[1663]{
   GP1:
	UF : 0, UT : 6,		CONFIG : 'N U T, 0, 0, 0',
	X =  344.485  mm,	Y =   -86.973  mm,	Z =   -263.039  mm,
	W =  90.000 deg,	P =   0.000 deg,	R =   90.000 deg
};
P[1664]{
   GP1:
	UF : 0, UT : 6,		CONFIG : 'N U T, 0, 0, 0',
	X =  343.554  mm,	Y =   -87.548  mm,	Z =   -263.129  mm,
	W =  90.000 deg,	P =   0.000 deg,	R =   90.000 deg
};
P[1665]{
   GP1:
	UF : 0, UT : 6,		CONFIG : 'N U T, 0, 0, 0',
	X =  342.835  mm,	Y =   -87.827  mm,	Z =   -262.797  mm,
	W =  90.000 deg,	P =   0.000 deg,	R =   90.000 deg
};
P[1666]{
   GP1:
	UF : 0, UT : 6,		CONFIG : 'N U T, 0, 0, 0',
	X =  341.759  mm,	Y =   -88.439  mm,	Z =   -262.778  mm,
	W =  90.000 deg,	P =   0.000 deg,	R =   90.000 deg
};
P[1667]{
   GP1:
	UF : 0, UT : 6,		CONFIG : 'N U T, 0, 0, 0',
	X =  340.015  mm,	Y =   -89.510  mm,	Z =   -262.931  mm,
	W =  90.000 deg,	P =   0.000 deg,	R =   90.000 deg
};
P[1668]{
   GP1:
	UF : 0, UT : 6,		CONFIG : 'N U T, 0, 0, 0',
	X =  339.049  mm,	Y =   -90.182  mm,	Z =   -263.210  mm,
	W =  90.000 deg,	P =   0.000 deg,	R =   90.000 deg
};
P[1669]{
   GP1:
	UF : 0, UT : 6,		CONFIG : 'N U T, 0, 0, 0',
	X =  337.699  mm,	Y =   -90.917  mm,	Z =   -263.101  mm,
	W =  90.000 deg,	P =   0.000 deg,	R =   90.000 deg
};
P[1670]{
   GP1:
	UF : 0, UT : 6,		CONFIG : 'N U T, 0, 0, 0',
	X =  336.231  mm,	Y =   -91.639  mm,	Z =   -262.796  mm,
	W =  90.000 deg,	P =   0.000 deg,	R =   90.000 deg
};
P[1671]{
   GP1:
	UF : 0, UT : 6,		CONFIG : 'N U T, 0, 0, 0',
	X =  334.711  mm,	Y =   -92.639  mm,	Z =   -263.093  mm,
	W =  90.000 deg,	P =   0.000 deg,	R =   90.000 deg
};
P[1672]{
   GP1:
	UF : 0, UT : 6,		CONFIG : 'N U T, 0, 0, 0',
	X =  333.809  mm,	Y =   -93.158  mm,	Z =   -263.088  mm,
	W =  90.000 deg,	P =   0.000 deg,	R =   90.000 deg
};
P[1673]{
   GP1:
	UF : 0, UT : 6,		CONFIG : 'N U T, 0, 0, 0',
	X =  333.022  mm,	Y =   -93.520  mm,	Z =   -262.865  mm,
	W =  90.000 deg,	P =   0.000 deg,	R =   90.000 deg
};
P[1674]{
   GP1:
	UF : 0, UT : 6,		CONFIG : 'N U T, 0, 0, 0',
	X =  331.976  mm,	Y =   -94.207  mm,	Z =   -263.065  mm,
	W =  90.000 deg,	P =   0.000 deg,	R =   90.000 deg
};
P[1675]{
   GP1:
	UF : 0, UT : 6,		CONFIG : 'N U T, 0, 0, 0',
	X =  330.323  mm,	Y =   -95.175  mm,	Z =   -263.098  mm,
	W =  90.000 deg,	P =   0.000 deg,	R =   90.000 deg
};
P[1676]{
   GP1:
	UF : 0, UT : 6,		CONFIG : 'N U T, 0, 0, 0',
	X =  329.069  mm,	Y =   -95.782  mm,	Z =   -262.815  mm,
	W =  90.000 deg,	P =   0.000 deg,	R =   90.000 deg
};
P[1677]{
   GP1:
	UF : 0, UT : 6,		CONFIG : 'N U T, 0, 0, 0',
	X =  326.943  mm,	Y =   -97.171  mm,	Z =   -263.208  mm,
	W =  90.000 deg,	P =   0.000 deg,	R =   90.000 deg
};
P[1678]{
   GP1:
	UF : 0, UT : 6,		CONFIG : 'N U T, 0, 0, 0',
	X =  325.490  mm,	Y =   -97.831  mm,	Z =   -262.774  mm,
	W =  90.000 deg,	P =   0.000 deg,	R =   90.000 deg
};
P[1679]{
   GP1:
	UF : 0, UT : 6,		CONFIG : 'N U T, 0, 0, 0',
	X =  323.252  mm,	Y =   -99.162  mm,	Z =   -262.866  mm,
	W =  90.000 deg,	P =   0.000 deg,	R =   90.000 deg
};
P[1680]{
   GP1:
	UF : 0, UT : 6,		CONFIG : 'N U T, 0, 0, 0',
	X =  321.894  mm,	Y =   -100.065  mm,	Z =   -263.156  mm,
	W =  90.000 deg,	P =   0.000 deg,	R =   90.000 deg
};
P[1681]{
   GP1:
	UF : 0, UT : 6,		CONFIG : 'N U T, 0, 0, 0',
	X =  320.688  mm,	Y =   -100.663  mm,	Z =   -262.917  mm,
	W =  90.000 deg,	P =   0.000 deg,	R =   90.000 deg
};
P[1682]{
   GP1:
	UF : 0, UT : 6,		CONFIG : 'N U T, 0, 0, 0',
	X =  318.864  mm,	Y =   -101.718  mm,	Z =   -262.920  mm,
	W =  90.000 deg,	P =   0.000 deg,	R =   90.000 deg
};
P[1683]{
   GP1:
	UF : 0, UT : 6,		CONFIG : 'N U T, 0, 0, 0',
	X =  315.976  mm,	Y =   -103.519  mm,	Z =   -263.243  mm,
	W =  90.000 deg,	P =   0.000 deg,	R =   90.000 deg
};
P[1684]{
   GP1:
	UF : 0, UT : 6,		CONFIG : 'N U T, 0, 0, 0',
	X =  314.089  mm,	Y =   -104.563  mm,	Z =   -263.137  mm,
	W =  90.000 deg,	P =   0.000 deg,	R =   90.000 deg
};
P[1685]{
   GP1:
	UF : 0, UT : 6,		CONFIG : 'N U T, 0, 0, 0',
	X =  313.251  mm,	Y =   -105.011  mm,	Z =   -263.048  mm,
	W =  90.000 deg,	P =   0.000 deg,	R =   90.000 deg
};
P[1686]{
   GP1:
	UF : 0, UT : 6,		CONFIG : 'N U T, 0, 0, 0',
	X =  312.185  mm,	Y =   -105.686  mm,	Z =   -263.193  mm,
	W =  90.000 deg,	P =   0.000 deg,	R =   90.000 deg
};
P[1687]{
   GP1:
	UF : 0, UT : 6,		CONFIG : 'N U T, 0, 0, 0',
	X =  310.724  mm,	Y =   -106.490  mm,	Z =   -263.098  mm,
	W =  90.000 deg,	P =   0.000 deg,	R =   90.000 deg
};
P[1688]{
   GP1:
	UF : 0, UT : 6,		CONFIG : 'N U T, 0, 0, 0',
	X =  309.152  mm,	Y =   -107.266  mm,	Z =   -262.777  mm,
	W =  90.000 deg,	P =   0.000 deg,	R =   90.000 deg
};
P[1689]{
   GP1:
	UF : 0, UT : 6,		CONFIG : 'N U T, 0, 0, 0',
	X =  305.669  mm,	Y =   -109.310  mm,	Z =   -262.856  mm,
	W =  90.000 deg,	P =   0.000 deg,	R =   90.000 deg
};
P[1690]{
   GP1:
	UF : 0, UT : 6,		CONFIG : 'N U T, 0, 0, 0',
	X =  304.829  mm,	Y =   -109.910  mm,	Z =   -263.136  mm,
	W =  90.000 deg,	P =   0.000 deg,	R =   90.000 deg
};
P[1691]{
   GP1:
	UF : 0, UT : 6,		CONFIG : 'N U T, 0, 0, 0',
	X =  301.982  mm,	Y =   -111.599  mm,	Z =   -263.244  mm,
	W =  90.000 deg,	P =   0.000 deg,	R =   90.000 deg
};
P[1692]{
   GP1:
	UF : 0, UT : 6,		CONFIG : 'N U T, 0, 0, 0',
	X =  301.170  mm,	Y =   -112.024  mm,	Z =   -263.138  mm,
	W =  90.000 deg,	P =   0.000 deg,	R =   90.000 deg
};
P[1693]{
   GP1:
	UF : 0, UT : 6,		CONFIG : 'N U T, 0, 0, 0',
	X =  299.432  mm,	Y =   -112.871  mm,	Z =   -262.759  mm,
	W =  90.000 deg,	P =   0.000 deg,	R =   90.000 deg
};
P[1694]{
   GP1:
	UF : 0, UT : 6,		CONFIG : 'N U T, 0, 0, 0',
	X =  297.721  mm,	Y =   -114.012  mm,	Z =   -263.130  mm,
	W =  90.000 deg,	P =   0.000 deg,	R =   90.000 deg
};
P[1695]{
   GP1:
	UF : 0, UT : 6,		CONFIG : 'N U T, 0, 0, 0',
	X =  296.491  mm,	Y =   -114.639  mm,	Z =   -262.929  mm,
	W =  90.000 deg,	P =   0.000 deg,	R =   90.000 deg
};
P[1696]{
   GP1:
	UF : 0, UT : 6,		CONFIG : 'N U T, 0, 0, 0',
	X =  293.957  mm,	Y =   -116.235  mm,	Z =   -263.252  mm,
	W =  90.000 deg,	P =   0.000 deg,	R =   90.000 deg
};
P[1697]{
   GP1:
	UF : 0, UT : 6,		CONFIG : 'N U T, 0, 0, 0',
	X =  291.387  mm,	Y =   -117.594  mm,	Z =   -262.947  mm,
	W =  90.000 deg,	P =   0.000 deg,	R =   90.000 deg
};
P[1698]{
   GP1:
	UF : 0, UT : 6,		CONFIG : 'N U T, 0, 0, 0',
	X =  290.527  mm,	Y =   -118.150  mm,	Z =   -263.093  mm,
	W =  90.000 deg,	P =   0.000 deg,	R =   90.000 deg
};
P[1699]{
   GP1:
	UF : 0, UT : 6,		CONFIG : 'N U T, 0, 0, 0',
	X =  289.546  mm,	Y =   -118.587  mm,	Z =   -262.779  mm,
	W =  90.000 deg,	P =   0.000 deg,	R =   90.000 deg
};
P[1700]{
   GP1:
	UF : 0, UT : 6,		CONFIG : 'N U T, 0, 0, 0',
	X =  288.081  mm,	Y =   -119.605  mm,	Z =   -263.195  mm,
	W =  90.000 deg,	P =   0.000 deg,	R =   90.000 deg
};
P[1701]{
   GP1:
	UF : 0, UT : 6,		CONFIG : 'N U T, 0, 0, 0',
	X =  287.043  mm,	Y =   -120.189  mm,	Z =   -263.157  mm,
	W =  90.000 deg,	P =   0.000 deg,	R =   90.000 deg
};
P[1702]{
   GP1:
	UF : 0, UT : 6,		CONFIG : 'N U T, 0, 0, 0',
	X =  285.831  mm,	Y =   -120.824  mm,	Z =   -263.002  mm,
	W =  90.000 deg,	P =   0.000 deg,	R =   90.000 deg
};
P[1703]{
   GP1:
	UF : 0, UT : 6,		CONFIG : 'N U T, 0, 0, 0',
	X =  284.506  mm,	Y =   -121.617  mm,	Z =   -263.068  mm,
	W =  90.000 deg,	P =   0.000 deg,	R =   90.000 deg
};
P[1704]{
   GP1:
	UF : 0, UT : 6,		CONFIG : 'N U T, 0, 0, 0',
	X =  283.585  mm,	Y =   -122.047  mm,	Z =   -262.825  mm,
	W =  90.000 deg,	P =   0.000 deg,	R =   90.000 deg
};
P[1705]{
   GP1:
	UF : 0, UT : 6,		CONFIG : 'N U T, 0, 0, 0',
	X =  282.197  mm,	Y =   -122.934  mm,	Z =   -263.031  mm,
	W =  90.000 deg,	P =   0.000 deg,	R =   90.000 deg
};
P[1706]{
   GP1:
	UF : 0, UT : 6,		CONFIG : 'N U T, 0, 0, 0',
	X =  280.740  mm,	Y =   -123.742  mm,	Z =   -262.948  mm,
	W =  90.000 deg,	P =   0.000 deg,	R =   90.000 deg
};
P[1707]{
   GP1:
	UF : 0, UT : 6,		CONFIG : 'N U T, 0, 0, 0',
	X =  279.975  mm,	Y =   -124.131  mm,	Z =   -262.823  mm,
	W =  90.000 deg,	P =   0.000 deg,	R =   90.000 deg
};
P[1708]{
   GP1:
	UF : 0, UT : 6,		CONFIG : 'N U T, 0, 0, 0',
	X =  279.252  mm,	Y =   -124.687  mm,	Z =   -263.158  mm,
	W =  90.000 deg,	P =   0.000 deg,	R =   90.000 deg
};
P[1709]{
   GP1:
	UF : 0, UT : 6,		CONFIG : 'N U T, 0, 0, 0',
	X =  277.334  mm,	Y =   -125.698  mm,	Z =   -262.923  mm,
	W =  90.000 deg,	P =   0.000 deg,	R =   90.000 deg
};
P[1710]{
   GP1:
	UF : 0, UT : 6,		CONFIG : 'N U T, 0, 0, 0',
	X =  273.592  mm,	Y =   -127.990  mm,	Z =   -263.243  mm,
	W =  90.000 deg,	P =   0.000 deg,	R =   90.000 deg
};
P[1711]{
   GP1:
	UF : 0, UT : 6,		CONFIG : 'N U T, 0, 0, 0',
	X =  272.211  mm,	Y =   -128.792  mm,	Z =   -263.252  mm,
	W =  90.000 deg,	P =   0.000 deg,	R =   90.000 deg
};
P[1712]{
   GP1:
	UF : 0, UT : 6,		CONFIG : 'N U T, 0, 0, 0',
	X =  270.857  mm,	Y =   -129.489  mm,	Z =   -263.048  mm,
	W =  90.000 deg,	P =   0.000 deg,	R =   90.000 deg
};
P[1713]{
   GP1:
	UF : 0, UT : 6,		CONFIG : 'N U T, 0, 0, 0',
	X =  268.967  mm,	Y =   -130.611  mm,	Z =   -263.122  mm,
	W =  90.000 deg,	P =   0.000 deg,	R =   90.000 deg
};
P[1714]{
   GP1:
	UF : 0, UT : 6,		CONFIG : 'N U T, 0, 0, 0',
	X =  267.609  mm,	Y =   -131.412  mm,	Z =   -263.165  mm,
	W =  90.000 deg,	P =   0.000 deg,	R =   90.000 deg
};
P[1715]{
   GP1:
	UF : 0, UT : 6,		CONFIG : 'N U T, 0, 0, 0',
	X =  266.120  mm,	Y =   -132.243  mm,	Z =   -263.095  mm,
	W =  90.000 deg,	P =   0.000 deg,	R =   90.000 deg
};
P[1716]{
   GP1:
	UF : 0, UT : 6,		CONFIG : 'N U T, 0, 0, 0',
	X =  259.164  mm,	Y =   -136.132  mm,	Z =   -262.783  mm,
	W =  90.000 deg,	P =   0.000 deg,	R =   90.000 deg
};
P[1717]{
   GP1:
	UF : 0, UT : 6,		CONFIG : 'N U T, 0, 0, 0',
	X =  257.968  mm,	Y =   -137.004  mm,	Z =   -263.226  mm,
	W =  90.000 deg,	P =   0.000 deg,	R =   90.000 deg
};
P[1718]{
   GP1:
	UF : 0, UT : 6,		CONFIG : 'N U T, 0, 0, 0',
	X =  256.016  mm,	Y =   -138.085  mm,	Z =   -263.113  mm,
	W =  90.000 deg,	P =   0.000 deg,	R =   90.000 deg
};
P[1719]{
   GP1:
	UF : 0, UT : 6,		CONFIG : 'N U T, 0, 0, 0',
	X =  254.118  mm,	Y =   -139.177  mm,	Z =   -263.102  mm,
	W =  90.000 deg,	P =   0.000 deg,	R =   90.000 deg
};
P[1720]{
   GP1:
	UF : 0, UT : 6,		CONFIG : 'N U T, 0, 0, 0',
	X =  253.205  mm,	Y =   -139.747  mm,	Z =   -263.209  mm,
	W =  90.000 deg,	P =   0.000 deg,	R =   90.000 deg
};
P[1721]{
   GP1:
	UF : 0, UT : 6,		CONFIG : 'N U T, 0, 0, 0',
	X =  252.371  mm,	Y =   -140.211  mm,	Z =   -263.164  mm,
	W =  90.000 deg,	P =   0.000 deg,	R =   90.000 deg
};
P[1722]{
   GP1:
	UF : 0, UT : 6,		CONFIG : 'N U T, 0, 0, 0',
	X =  251.565  mm,	Y =   -140.562  mm,	Z =   -262.889  mm,
	W =  90.000 deg,	P =   0.000 deg,	R =   90.000 deg
};
P[1723]{
   GP1:
	UF : 0, UT : 6,		CONFIG : 'N U T, 0, 0, 0',
	X =  250.671  mm,	Y =   -141.080  mm,	Z =   -262.890  mm,
	W =  90.000 deg,	P =   0.000 deg,	R =   90.000 deg
};
P[1724]{
   GP1:
	UF : 0, UT : 6,		CONFIG : 'N U T, 0, 0, 0',
	X =  249.050  mm,	Y =   -142.054  mm,	Z =   -262.986  mm,
	W =  90.000 deg,	P =   0.000 deg,	R =   90.000 deg
};
P[1725]{
   GP1:
	UF : 0, UT : 6,		CONFIG : 'N U T, 0, 0, 0',
	X =  246.004  mm,	Y =   -143.884  mm,	Z =   -263.157  mm,
	W =  90.000 deg,	P =   0.000 deg,	R =   90.000 deg
};
P[1726]{
   GP1:
	UF : 0, UT : 6,		CONFIG : 'N U T, 0, 0, 0',
	X =  244.737  mm,	Y =   -144.574  mm,	Z =   -263.057  mm,
	W =  90.000 deg,	P =   0.000 deg,	R =   90.000 deg
};
P[1727]{
   GP1:
	UF : 0, UT : 6,		CONFIG : 'N U T, 0, 0, 0',
	X =  243.016  mm,	Y =   -145.506  mm,	Z =   -262.906  mm,
	W =  90.000 deg,	P =   0.000 deg,	R =   90.000 deg
};
P[1728]{
   GP1:
	UF : 0, UT : 6,		CONFIG : 'N U T, 0, 0, 0',
	X =  237.049  mm,	Y =   -149.015  mm,	Z =   -263.062  mm,
	W =  90.000 deg,	P =   0.000 deg,	R =   90.000 deg
};
P[1729]{
   GP1:
	UF : 0, UT : 6,		CONFIG : 'N U T, 0, 0, 0',
	X =  236.158  mm,	Y =   -149.532  mm,	Z =   -263.067  mm,
	W =  90.000 deg,	P =   0.000 deg,	R =   90.000 deg
};
P[1730]{
   GP1:
	UF : 0, UT : 6,		CONFIG : 'N U T, 0, 0, 0',
	X =  235.168  mm,	Y =   -150.052  mm,	Z =   -262.939  mm,
	W =  90.000 deg,	P =   0.000 deg,	R =   90.000 deg
};
P[1731]{
   GP1:
	UF : 0, UT : 6,		CONFIG : 'N U T, 0, 0, 0',
	X =  233.710  mm,	Y =   -150.878  mm,	Z =   -262.904  mm,
	W =  90.000 deg,	P =   0.000 deg,	R =   90.000 deg
};
P[1732]{
   GP1:
	UF : 0, UT : 6,		CONFIG : 'N U T, 0, 0, 0',
	X =  231.592  mm,	Y =   -152.084  mm,	Z =   -262.860  mm,
	W =  90.000 deg,	P =   0.000 deg,	R =   90.000 deg
};
P[1733]{
   GP1:
	UF : 0, UT : 6,		CONFIG : 'N U T, 0, 0, 0',
	X =  230.880  mm,	Y =   -152.562  mm,	Z =   -263.025  mm,
	W =  90.000 deg,	P =   0.000 deg,	R =   90.000 deg
};
P[1734]{
   GP1:
	UF : 0, UT : 6,		CONFIG : 'N U T, 0, 0, 0',
	X =  228.646  mm,	Y =   -153.743  mm,	Z =   -262.760  mm,
	W =  90.000 deg,	P =   0.000 deg,	R =   90.000 deg
};
P[1735]{
   GP1:
	UF : 0, UT : 6,		CONFIG : 'N U T, 0, 0, 0',
	X =  227.326  mm,	Y =   -154.523  mm,	Z =   -262.803  mm,
	W =  90.000 deg,	P =   0.000 deg,	R =   90.000 deg
};
P[1736]{
   GP1:
	UF : 0, UT : 6,		CONFIG : 'N U T, 0, 0, 0',
	X =  226.714  mm,	Y =   -154.936  mm,	Z =   -262.949  mm,
	W =  90.000 deg,	P =   0.000 deg,	R =   90.000 deg
};
P[1737]{
   GP1:
	UF : 0, UT : 6,		CONFIG : 'N U T, 0, 0, 0',
	X =  225.606  mm,	Y =   -155.623  mm,	Z =   -263.064  mm,
	W =  90.000 deg,	P =   0.000 deg,	R =   90.000 deg
};
P[1738]{
   GP1:
	UF : 0, UT : 6,		CONFIG : 'N U T, 0, 0, 0',
	X =  224.512  mm,	Y =   -156.209  mm,	Z =   -262.954  mm,
	W =  90.000 deg,	P =   0.000 deg,	R =   90.000 deg
};
P[1739]{
   GP1:
	UF : 0, UT : 6,		CONFIG : 'N U T, 0, 0, 0',
	X =  222.701  mm,	Y =   -157.304  mm,	Z =   -263.070  mm,
	W =  90.000 deg,	P =   0.000 deg,	R =   90.000 deg
};
P[1740]{
   GP1:
	UF : 0, UT : 6,		CONFIG : 'N U T, 0, 0, 0',
	X =  221.498  mm,	Y =   -158.029  mm,	Z =   -263.146  mm,
	W =  90.000 deg,	P =   0.000 deg,	R =   90.000 deg
};
P[1741]{
   GP1:
	UF : 0, UT : 6,		CONFIG : 'N U T, 0, 0, 0',
	X =  218.854  mm,	Y =   -159.452  mm,	Z =   -262.894  mm,
	W =  90.000 deg,	P =   0.000 deg,	R =   90.000 deg
};
P[1742]{
   GP1:
	UF : 0, UT : 6,		CONFIG : 'N U T, 0, 0, 0',
	X =  217.653  mm,	Y =   -160.144  mm,	Z =   -262.891  mm,
	W =  90.000 deg,	P =   0.000 deg,	R =   90.000 deg
};
P[1743]{
   GP1:
	UF : 0, UT : 6,		CONFIG : 'N U T, 0, 0, 0',
	X =  216.022  mm,	Y =   -161.179  mm,	Z =   -263.115  mm,
	W =  90.000 deg,	P =   0.000 deg,	R =   90.000 deg
};
P[1744]{
   GP1:
	UF : 0, UT : 6,		CONFIG : 'N U T, 0, 0, 0',
	X =  215.074  mm,	Y =   -161.640  mm,	Z =   -262.908  mm,
	W =  90.000 deg,	P =   0.000 deg,	R =   90.000 deg
};
P[1745]{
   GP1:
	UF : 0, UT : 6,		CONFIG : 'N U T, 0, 0, 0',
	X =  214.042  mm,	Y =   -162.336  mm,	Z =   -263.150  mm,
	W =  90.000 deg,	P =   0.000 deg,	R =   90.000 deg
};
P[1746]{
   GP1:
	UF : 0, UT : 6,		CONFIG : 'N U T, 0, 0, 0',
	X =  213.087  mm,	Y =   -162.820  mm,	Z =   -262.988  mm,
	W =  90.000 deg,	P =   0.000 deg,	R =   90.000 deg
};
P[1747]{
   GP1:
	UF : 0, UT : 6,		CONFIG : 'N U T, 0, 0, 0',
	X =  211.694  mm,	Y =   -163.603  mm,	Z =   -262.934  mm,
	W =  90.000 deg,	P =   0.000 deg,	R =   90.000 deg
};
P[1748]{
   GP1:
	UF : 0, UT : 6,		CONFIG : 'N U T, 0, 0, 0',
	X =  209.063  mm,	Y =   -165.109  mm,	Z =   -262.906  mm,
	W =  90.000 deg,	P =   0.000 deg,	R =   90.000 deg
};
P[1749]{
   GP1:
	UF : 0, UT : 6,		CONFIG : 'N U T, 0, 0, 0',
	X =  206.490  mm,	Y =   -166.602  mm,	Z =   -262.920  mm,
	W =  90.000 deg,	P =   0.000 deg,	R =   90.000 deg
};
P[1750]{
   GP1:
	UF : 0, UT : 6,		CONFIG : 'N U T, 0, 0, 0',
	X =  205.654  mm,	Y =   -167.081  mm,	Z =   -262.913  mm,
	W =  90.000 deg,	P =   0.000 deg,	R =   90.000 deg
};
P[1751]{
   GP1:
	UF : 0, UT : 6,		CONFIG : 'N U T, 0, 0, 0',
	X =  204.571  mm,	Y =   -167.716  mm,	Z =   -262.935  mm,
	W =  90.000 deg,	P =   0.000 deg,	R =   90.000 deg
};
P[1752]{
   GP1:
	UF : 0, UT : 6,		CONFIG : 'N U T, 0, 0, 0',
	X =  202.241  mm,	Y =   -169.185  mm,	Z =   -263.236  mm,
	W =  90.000 deg,	P =   0.000 deg,	R =   90.000 deg
};
P[1753]{
   GP1:
	UF : 0, UT : 6,		CONFIG : 'N U T, 0, 0, 0',
	X =  201.452  mm,	Y =   -169.539  mm,	Z =   -262.989  mm,
	W =  90.000 deg,	P =   0.000 deg,	R =   90.000 deg
};
P[1754]{
   GP1:
	UF : 0, UT : 6,		CONFIG : 'N U T, 0, 0, 0',
	X =  200.519  mm,	Y =   -170.018  mm,	Z =   -262.846  mm,
	W =  90.000 deg,	P =   0.000 deg,	R =   90.000 deg
};
P[1755]{
   GP1:
	UF : 0, UT : 6,		CONFIG : 'N U T, 0, 0, 0',
	X =  199.773  mm,	Y =   -170.574  mm,	Z =   -263.148  mm,
	W =  90.000 deg,	P =   0.000 deg,	R =   90.000 deg
};
P[1756]{
   GP1:
	UF : 0, UT : 6,		CONFIG : 'N U T, 0, 0, 0',
	X =  199.121  mm,	Y =   -170.922  mm,	Z =   -263.079  mm,
	W =  90.000 deg,	P =   0.000 deg,	R =   90.000 deg
};
P[1757]{
   GP1:
	UF : 0, UT : 6,		CONFIG : 'N U T, 0, 0, 0',
	X =  195.900  mm,	Y =   -172.707  mm,	Z =   -262.899  mm,
	W =  90.000 deg,	P =   0.000 deg,	R =   90.000 deg
};
P[1758]{
   GP1:
	UF : 0, UT : 6,		CONFIG : 'N U T, 0, 0, 0',
	X =  194.569  mm,	Y =   -173.584  mm,	Z =   -263.162  mm,
	W =  90.000 deg,	P =   0.000 deg,	R =   90.000 deg
};
P[1759]{
   GP1:
	UF : 0, UT : 6,		CONFIG : 'N U T, 0, 0, 0',
	X =  190.956  mm,	Y =   -175.692  mm,	Z =   -263.214  mm,
	W =  90.000 deg,	P =   0.000 deg,	R =   90.000 deg
};
P[1760]{
   GP1:
	UF : 0, UT : 6,		CONFIG : 'N U T, 0, 0, 0',
	X =  186.838  mm,	Y =   -178.008  mm,	Z =   -263.066  mm,
	W =  90.000 deg,	P =   0.000 deg,	R =   90.000 deg
};
P[1761]{
   GP1:
	UF : 0, UT : 6,		CONFIG : 'N U T, 0, 0, 0',
	X =  186.214  mm,	Y =   -178.377  mm,	Z =   -263.086  mm,
	W =  90.000 deg,	P =   0.000 deg,	R =   90.000 deg
};
P[1762]{
   GP1:
	UF : 0, UT : 6,		CONFIG : 'N U T, 0, 0, 0',
	X =  185.493  mm,	Y =   -178.781  mm,	Z =   -263.054  mm,
	W =  90.000 deg,	P =   0.000 deg,	R =   90.000 deg
};
P[1763]{
   GP1:
	UF : 0, UT : 6,		CONFIG : 'N U T, 0, 0, 0',
	X =  184.192  mm,	Y =   -179.597  mm,	Z =   -263.216  mm,
	W =  90.000 deg,	P =   0.000 deg,	R =   90.000 deg
};
P[1764]{
   GP1:
	UF : 0, UT : 6,		CONFIG : 'N U T, 0, 0, 0',
	X =  178.896  mm,	Y =   -182.604  mm,	Z =   -263.091  mm,
	W =  90.000 deg,	P =   0.000 deg,	R =   90.000 deg
};
P[1765]{
   GP1:
	UF : 0, UT : 6,		CONFIG : 'N U T, 0, 0, 0',
	X =  177.201  mm,	Y =   -183.625  mm,	Z =   -263.193  mm,
	W =  90.000 deg,	P =   0.000 deg,	R =   90.000 deg
};
P[1766]{
   GP1:
	UF : 0, UT : 6,		CONFIG : 'N U T, 0, 0, 0',
	X =  176.060  mm,	Y =   -184.214  mm,	Z =   -263.025  mm,
	W =  90.000 deg,	P =   0.000 deg,	R =   90.000 deg
};
P[1767]{
   GP1:
	UF : 0, UT : 6,		CONFIG : 'N U T, 0, 0, 0',
	X =  173.664  mm,	Y =   -185.660  mm,	Z =   -263.176  mm,
	W =  90.000 deg,	P =   0.000 deg,	R =   90.000 deg
};
P[1768]{
   GP1:
	UF : 0, UT : 6,		CONFIG : 'N U T, 0, 0, 0',
	X =  171.586  mm,	Y =   -186.830  mm,	Z =   -263.103  mm,
	W =  90.000 deg,	P =   0.000 deg,	R =   90.000 deg
};
P[1769]{
   GP1:
	UF : 0, UT : 6,		CONFIG : 'N U T, 0, 0, 0',
	X =  170.220  mm,	Y =   -187.598  mm,	Z =   -263.052  mm,
	W =  90.000 deg,	P =   0.000 deg,	R =   90.000 deg
};
P[1770]{
   GP1:
	UF : 0, UT : 6,		CONFIG : 'N U T, 0, 0, 0',
	X =  169.063  mm,	Y =   -188.324  mm,	Z =   -263.191  mm,
	W =  90.000 deg,	P =   0.000 deg,	R =   90.000 deg
};
P[1771]{
   GP1:
	UF : 0, UT : 6,		CONFIG : 'N U T, 0, 0, 0',
	X =  167.597  mm,	Y =   -189.100  mm,	Z =   -263.021  mm,
	W =  90.000 deg,	P =   0.000 deg,	R =   90.000 deg
};
P[1772]{
   GP1:
	UF : 0, UT : 6,		CONFIG : 'N U T, 0, 0, 0',
	X =  166.470  mm,	Y =   -189.828  mm,	Z =   -263.210  mm,
	W =  90.000 deg,	P =   0.000 deg,	R =   90.000 deg
};
P[1773]{
   GP1:
	UF : 0, UT : 6,		CONFIG : 'N U T, 0, 0, 0',
	X =  162.560  mm,	Y =   -192.088  mm,	Z =   -263.216  mm,
	W =  90.000 deg,	P =   0.000 deg,	R =   90.000 deg
};
P[1774]{
   GP1:
	UF : 0, UT : 6,		CONFIG : 'N U T, 0, 0, 0',
	X =  161.858  mm,	Y =   -192.458  mm,	Z =   -263.131  mm,
	W =  90.000 deg,	P =   0.000 deg,	R =   90.000 deg
};
P[1775]{
   GP1:
	UF : 0, UT : 6,		CONFIG : 'N U T, 0, 0, 0',
	X =  160.866  mm,	Y =   -193.012  mm,	Z =   -263.087  mm,
	W =  90.000 deg,	P =   0.000 deg,	R =   90.000 deg
};
P[1776]{
   GP1:
	UF : 0, UT : 6,		CONFIG : 'N U T, 0, 0, 0',
	X =  159.720  mm,	Y =   -193.599  mm,	Z =   -262.904  mm,
	W =  90.000 deg,	P =   0.000 deg,	R =   90.000 deg
};
P[1777]{
   GP1:
	UF : 0, UT : 6,		CONFIG : 'N U T, 0, 0, 0',
	X =  158.466  mm,	Y =   -194.366  mm,	Z =   -263.007  mm,
	W =  90.000 deg,	P =   0.000 deg,	R =   90.000 deg
};
P[1778]{
   GP1:
	UF : 0, UT : 6,		CONFIG : 'N U T, 0, 0, 0',
	X =  157.551  mm,	Y =   -194.931  mm,	Z =   -263.097  mm,
	W =  90.000 deg,	P =   0.000 deg,	R =   90.000 deg
};
P[1779]{
   GP1:
	UF : 0, UT : 6,		CONFIG : 'N U T, 0, 0, 0',
	X =  155.718  mm,	Y =   -196.042  mm,	Z =   -263.225  mm,
	W =  90.000 deg,	P =   0.000 deg,	R =   90.000 deg
};
P[1780]{
   GP1:
	UF : 0, UT : 6,		CONFIG : 'N U T, 0, 0, 0',
	X =  154.767  mm,	Y =   -196.421  mm,	Z =   -262.812  mm,
	W =  90.000 deg,	P =   0.000 deg,	R =   90.000 deg
};
P[1781]{
   GP1:
	UF : 0, UT : 6,		CONFIG : 'N U T, 0, 0, 0',
	X =  153.577  mm,	Y =   -197.117  mm,	Z =   -262.834  mm,
	W =  90.000 deg,	P =   0.000 deg,	R =   90.000 deg
};
P[1782]{
   GP1:
	UF : 0, UT : 6,		CONFIG : 'N U T, 0, 0, 0',
	X =  151.612  mm,	Y =   -198.422  mm,	Z =   -263.248  mm,
	W =  90.000 deg,	P =   0.000 deg,	R =   90.000 deg
};
P[1783]{
   GP1:
	UF : 0, UT : 6,		CONFIG : 'N U T, 0, 0, 0',
	X =  150.655  mm,	Y =   -198.957  mm,	Z =   -263.205  mm,
	W =  90.000 deg,	P =   0.000 deg,	R =   90.000 deg
};
P[1784]{
   GP1:
	UF : 0, UT : 6,		CONFIG : 'N U T, 0, 0, 0',
	X =  149.528  mm,	Y =   -199.433  mm,	Z =   -262.779  mm,
	W =  90.000 deg,	P =   0.000 deg,	R =   90.000 deg
};
P[1785]{
   GP1:
	UF : 0, UT : 6,		CONFIG : 'N U T, 0, 0, 0',
	X =  147.974  mm,	Y =   -200.413  mm,	Z =   -262.978  mm,
	W =  90.000 deg,	P =   0.000 deg,	R =   90.000 deg
};
P[1786]{
   GP1:
	UF : 0, UT : 6,		CONFIG : 'N U T, 0, 0, 0',
	X =  146.454  mm,	Y =   -201.317  mm,	Z =   -263.045  mm,
	W =  90.000 deg,	P =   0.000 deg,	R =   90.000 deg
};
P[1787]{
   GP1:
	UF : 0, UT : 6,		CONFIG : 'N U T, 0, 0, 0',
	X =  144.608  mm,	Y =   -202.336  mm,	Z =   -262.932  mm,
	W =  90.000 deg,	P =   0.000 deg,	R =   90.000 deg
};
P[1788]{
   GP1:
	UF : 0, UT : 6,		CONFIG : 'N U T, 0, 0, 0',
	X =  143.456  mm,	Y =   -202.997  mm,	Z =   -262.922  mm,
	W =  90.000 deg,	P =   0.000 deg,	R =   90.000 deg
};
P[1789]{
   GP1:
	UF : 0, UT : 6,		CONFIG : 'N U T, 0, 0, 0',
	X =  142.638  mm,	Y =   -203.508  mm,	Z =   -263.013  mm,
	W =  90.000 deg,	P =   0.000 deg,	R =   90.000 deg
};
P[1790]{
   GP1:
	UF : 0, UT : 6,		CONFIG : 'N U T, 0, 0, 0',
	X =  138.726  mm,	Y =   -205.729  mm,	Z =   -262.924  mm,
	W =  90.000 deg,	P =   0.000 deg,	R =   90.000 deg
};
P[1791]{
   GP1:
	UF : 0, UT : 6,		CONFIG : 'N U T, 0, 0, 0',
	X =  136.664  mm,	Y =   -206.957  mm,	Z =   -263.015  mm,
	W =  90.000 deg,	P =   0.000 deg,	R =   90.000 deg
};
P[1792]{
   GP1:
	UF : 0, UT : 6,		CONFIG : 'N U T, 0, 0, 0',
	X =  135.580  mm,	Y =   -207.494  mm,	Z =   -262.797  mm,
	W =  90.000 deg,	P =   0.000 deg,	R =   90.000 deg
};
P[1793]{
   GP1:
	UF : 0, UT : 6,		CONFIG : 'N U T, 0, 0, 0',
	X =  132.690  mm,	Y =   -209.185  mm,	Z =   -262.853  mm,
	W =  90.000 deg,	P =   0.000 deg,	R =   90.000 deg
};
P[1794]{
   GP1:
	UF : 0, UT : 6,		CONFIG : 'N U T, 0, 0, 0',
	X =  130.373  mm,	Y =   -210.533  mm,	Z =   -262.876  mm,
	W =  90.000 deg,	P =   0.000 deg,	R =   90.000 deg
};
P[1795]{
   GP1:
	UF : 0, UT : 6,		CONFIG : 'N U T, 0, 0, 0',
	X =  128.686  mm,	Y =   -211.619  mm,	Z =   -263.148  mm,
	W =  90.000 deg,	P =   0.000 deg,	R =   90.000 deg
};
P[1796]{
   GP1:
	UF : 0, UT : 6,		CONFIG : 'N U T, 0, 0, 0',
	X =  127.989  mm,	Y =   -211.944  mm,	Z =   -262.961  mm,
	W =  90.000 deg,	P =   0.000 deg,	R =   90.000 deg
};
P[1797]{
   GP1:
	UF : 0, UT : 6,		CONFIG : 'N U T, 0, 0, 0',
	X =  126.975  mm,	Y =   -212.507  mm,	Z =   -262.908  mm,
	W =  90.000 deg,	P =   0.000 deg,	R =   90.000 deg
};
P[1798]{
   GP1:
	UF : 0, UT : 6,		CONFIG : 'N U T, 0, 0, 0',
	X =  125.986  mm,	Y =   -213.046  mm,	Z =   -262.828  mm,
	W =  90.000 deg,	P =   0.000 deg,	R =   90.000 deg
};
P[1799]{
   GP1:
	UF : 0, UT : 6,		CONFIG : 'N U T, 0, 0, 0',
	X =  124.707  mm,	Y =   -213.883  mm,	Z =   -263.069  mm,
	W =  90.000 deg,	P =   0.000 deg,	R =   90.000 deg
};
P[1800]{
   GP1:
	UF : 0, UT : 6,		CONFIG : 'N U T, 0, 0, 0',
	X =  123.347  mm,	Y =   -214.635  mm,	Z =   -262.988  mm,
	W =  90.000 deg,	P =   0.000 deg,	R =   90.000 deg
};
P[1801]{
   GP1:
	UF : 0, UT : 6,		CONFIG : 'N U T, 0, 0, 0',
	X =  120.962  mm,	Y =   -216.099  mm,	Z =   -263.199  mm,
	W =  90.000 deg,	P =   0.000 deg,	R =   90.000 deg
};
P[1802]{
   GP1:
	UF : 0, UT : 6,		CONFIG : 'N U T, 0, 0, 0',
	X =  120.202  mm,	Y =   -216.547  mm,	Z =   -263.219  mm,
	W =  90.000 deg,	P =   0.000 deg,	R =   90.000 deg
};
P[1803]{
   GP1:
	UF : 0, UT : 6,		CONFIG : 'N U T, 0, 0, 0',
	X =  119.062  mm,	Y =   -217.107  mm,	Z =   -262.981  mm,
	W =  90.000 deg,	P =   0.000 deg,	R =   90.000 deg
};
P[1804]{
   GP1:
	UF : 0, UT : 6,		CONFIG : 'N U T, 0, 0, 0',
	X =  117.478  mm,	Y =   -215.670  mm,	Z =   -257.275  mm,
	W =  90.000 deg,	P =   0.000 deg,	R =   90.000 deg
};
P[1805]{
   GP1:
	UF : 0, UT : 6,		CONFIG : 'N U T, 0, 0, 0',
	X =  116.193  mm,	Y =   -216.368  mm,	Z =   -257.167  mm,
	W =  90.000 deg,	P =   0.000 deg,	R =   90.000 deg
};
P[1806]{
   GP1:
	UF : 0, UT : 6,		CONFIG : 'N U T, 0, 0, 0',
	X =  112.386  mm,	Y =   -218.593  mm,	Z =   -257.233  mm,
	W =  90.000 deg,	P =   0.000 deg,	R =   90.000 deg
};
P[1807]{
   GP1:
	UF : 0, UT : 6,		CONFIG : 'N U T, 0, 0, 0',
	X =  111.420  mm,	Y =   -219.177  mm,	Z =   -257.294  mm,
	W =  90.000 deg,	P =   0.000 deg,	R =   90.000 deg
};
P[1808]{
   GP1:
	UF : 0, UT : 6,		CONFIG : 'N U T, 0, 0, 0',
	X =  109.579  mm,	Y =   -220.099  mm,	Z =   -256.955  mm,
	W =  90.000 deg,	P =   0.000 deg,	R =   90.000 deg
};
P[1809]{
   GP1:
	UF : 0, UT : 6,		CONFIG : 'N U T, 0, 0, 0',
	X =  109.014  mm,	Y =   -220.546  mm,	Z =   -257.248  mm,
	W =  90.000 deg,	P =   0.000 deg,	R =   90.000 deg
};
P[1810]{
   GP1:
	UF : 0, UT : 6,		CONFIG : 'N U T, 0, 0, 0',
	X =  107.688  mm,	Y =   -221.257  mm,	Z =   -257.116  mm,
	W =  90.000 deg,	P =   0.000 deg,	R =   90.000 deg
};
P[1811]{
   GP1:
	UF : 0, UT : 6,		CONFIG : 'N U T, 0, 0, 0',
	X =  106.989  mm,	Y =   -221.700  mm,	Z =   -257.212  mm,
	W =  90.000 deg,	P =   0.000 deg,	R =   90.000 deg
};
P[1812]{
   GP1:
	UF : 0, UT : 6,		CONFIG : 'N U T, 0, 0, 0',
	X =  106.138  mm,	Y =   -222.220  mm,	Z =   -257.280  mm,
	W =  90.000 deg,	P =   0.000 deg,	R =   90.000 deg
};
P[1813]{
   GP1:
	UF : 0, UT : 6,		CONFIG : 'N U T, 0, 0, 0',
	X =  105.007  mm,	Y =   -222.900  mm,	Z =   -257.346  mm,
	W =  90.000 deg,	P =   0.000 deg,	R =   90.000 deg
};
P[1814]{
   GP1:
	UF : 0, UT : 6,		CONFIG : 'N U T, 0, 0, 0',
	X =  104.048  mm,	Y =   -223.449  mm,	Z =   -257.334  mm,
	W =  90.000 deg,	P =   0.000 deg,	R =   90.000 deg
};
P[1815]{
   GP1:
	UF : 0, UT : 6,		CONFIG : 'N U T, 0, 0, 0',
	X =  93.196  mm,	Y =   -229.569  mm,	Z =   -256.981  mm,
	W =  90.000 deg,	P =   0.000 deg,	R =   90.000 deg
};
P[1816]{
   GP1:
	UF : 0, UT : 6,		CONFIG : 'N U T, 0, 0, 0',
	X =  90.324  mm,	Y =   -231.361  mm,	Z =   -257.303  mm,
	W =  90.000 deg,	P =   0.000 deg,	R =   90.000 deg
};
P[1817]{
   GP1:
	UF : 0, UT : 6,		CONFIG : 'N U T, 0, 0, 0',
	X =  89.280  mm,	Y =   -231.937  mm,	Z =   -257.240  mm,
	W =  90.000 deg,	P =   0.000 deg,	R =   90.000 deg
};
P[1818]{
   GP1:
	UF : 0, UT : 6,		CONFIG : 'N U T, 0, 0, 0',
	X =  87.171  mm,	Y =   -233.135  mm,	Z =   -257.194  mm,
	W =  90.000 deg,	P =   0.000 deg,	R =   90.000 deg
};
P[1819]{
   GP1:
	UF : 0, UT : 6,		CONFIG : 'N U T, 0, 0, 0',
	X =  85.786  mm,	Y =   -233.829  mm,	Z =   -256.933  mm,
	W =  90.000 deg,	P =   0.000 deg,	R =   90.000 deg
};
P[1820]{
   GP1:
	UF : 0, UT : 6,		CONFIG : 'N U T, 0, 0, 0',
	X =  81.999  mm,	Y =   -236.157  mm,	Z =   -257.279  mm,
	W =  90.000 deg,	P =   0.000 deg,	R =   90.000 deg
};
P[1821]{
   GP1:
	UF : 0, UT : 6,		CONFIG : 'N U T, 0, 0, 0',
	X =  81.157  mm,	Y =   -236.604  mm,	Z =   -257.184  mm,
	W =  90.000 deg,	P =   0.000 deg,	R =   90.000 deg
};
P[1822]{
   GP1:
	UF : 0, UT : 6,		CONFIG : 'N U T, 0, 0, 0',
	X =  78.185  mm,	Y =   -238.302  mm,	Z =   -257.140  mm,
	W =  90.000 deg,	P =   0.000 deg,	R =   90.000 deg
};
P[1823]{
   GP1:
	UF : 0, UT : 6,		CONFIG : 'N U T, 0, 0, 0',
	X =  76.397  mm,	Y =   -239.378  mm,	Z =   -257.246  mm,
	W =  90.000 deg,	P =   0.000 deg,	R =   90.000 deg
};
P[1824]{
   GP1:
	UF : 0, UT : 6,		CONFIG : 'N U T, 0, 0, 0',
	X =  75.357  mm,	Y =   -239.865  mm,	Z =   -256.970  mm,
	W =  90.000 deg,	P =   0.000 deg,	R =   90.000 deg
};
P[1825]{
   GP1:
	UF : 0, UT : 6,		CONFIG : 'N U T, 0, 0, 0',
	X =  74.166  mm,	Y =   -240.629  mm,	Z =   -257.157  mm,
	W =  90.000 deg,	P =   0.000 deg,	R =   90.000 deg
};
P[1826]{
   GP1:
	UF : 0, UT : 6,		CONFIG : 'N U T, 0, 0, 0',
	X =  73.386  mm,	Y =   -241.153  mm,	Z =   -257.335  mm,
	W =  90.000 deg,	P =   0.000 deg,	R =   90.000 deg
};
P[1827]{
   GP1:
	UF : 0, UT : 6,		CONFIG : 'N U T, 0, 0, 0',
	X =  71.071  mm,	Y =   -242.487  mm,	Z =   -257.328  mm,
	W =  90.000 deg,	P =   0.000 deg,	R =   90.000 deg
};
P[1828]{
   GP1:
	UF : 0, UT : 6,		CONFIG : 'N U T, 0, 0, 0',
	X =  69.156  mm,	Y =   -243.560  mm,	Z =   -257.248  mm,
	W =  90.000 deg,	P =   0.000 deg,	R =   90.000 deg
};
P[1829]{
   GP1:
	UF : 0, UT : 6,		CONFIG : 'N U T, 0, 0, 0',
	X =  67.969  mm,	Y =   -244.248  mm,	Z =   -257.254  mm,
	W =  90.000 deg,	P =   0.000 deg,	R =   90.000 deg
};
P[1830]{
   GP1:
	UF : 0, UT : 6,		CONFIG : 'N U T, 0, 0, 0',
	X =  66.438  mm,	Y =   -244.990  mm,	Z =   -256.909  mm,
	W =  90.000 deg,	P =   0.000 deg,	R =   90.000 deg
};
P[1831]{
   GP1:
	UF : 0, UT : 6,		CONFIG : 'N U T, 0, 0, 0',
	X =  65.777  mm,	Y =   -245.449  mm,	Z =   -257.100  mm,
	W =  90.000 deg,	P =   0.000 deg,	R =   90.000 deg
};
P[1832]{
   GP1:
	UF : 0, UT : 6,		CONFIG : 'N U T, 0, 0, 0',
	X =  63.869  mm,	Y =   -246.668  mm,	Z =   -257.383  mm,
	W =  90.000 deg,	P =   0.000 deg,	R =   90.000 deg
};
P[1833]{
   GP1:
	UF : 0, UT : 6,		CONFIG : 'N U T, 0, 0, 0',
	X =  62.876  mm,	Y =   -247.215  mm,	Z =   -257.318  mm,
	W =  90.000 deg,	P =   0.000 deg,	R =   90.000 deg
};
P[1834]{
   GP1:
	UF : 0, UT : 6,		CONFIG : 'N U T, 0, 0, 0',
	X =  61.563  mm,	Y =   -247.903  mm,	Z =   -257.149  mm,
	W =  90.000 deg,	P =   0.000 deg,	R =   90.000 deg
};
P[1835]{
   GP1:
	UF : 0, UT : 6,		CONFIG : 'N U T, 0, 0, 0',
	X =  59.597  mm,	Y =   -249.041  mm,	Z =   -257.156  mm,
	W =  90.000 deg,	P =   0.000 deg,	R =   90.000 deg
};
P[1836]{
   GP1:
	UF : 0, UT : 6,		CONFIG : 'N U T, 0, 0, 0',
	X =  56.853  mm,	Y =   -250.696  mm,	Z =   -257.327  mm,
	W =  90.000 deg,	P =   0.000 deg,	R =   90.000 deg
};
P[1837]{
   GP1:
	UF : 0, UT : 6,		CONFIG : 'N U T, 0, 0, 0',
	X =  55.046  mm,	Y =   -251.626  mm,	Z =   -257.052  mm,
	W =  90.000 deg,	P =   0.000 deg,	R =   90.000 deg
};
P[1838]{
   GP1:
	UF : 0, UT : 6,		CONFIG : 'N U T, 0, 0, 0',
	X =  53.871  mm,	Y =   -252.330  mm,	Z =   -257.114  mm,
	W =  90.000 deg,	P =   0.000 deg,	R =   90.000 deg
};
P[1839]{
   GP1:
	UF : 0, UT : 6,		CONFIG : 'N U T, 0, 0, 0',
	X =  52.847  mm,	Y =   -252.971  mm,	Z =   -257.232  mm,
	W =  90.000 deg,	P =   0.000 deg,	R =   90.000 deg
};
P[1840]{
   GP1:
	UF : 0, UT : 6,		CONFIG : 'N U T, 0, 0, 0',
	X =  49.731  mm,	Y =   -254.832  mm,	Z =   -257.384  mm,
	W =  90.000 deg,	P =   0.000 deg,	R =   90.000 deg
};
P[1841]{
   GP1:
	UF : 0, UT : 6,		CONFIG : 'N U T, 0, 0, 0',
	X =  49.079  mm,	Y =   -255.138  mm,	Z =   -257.213  mm,
	W =  90.000 deg,	P =   0.000 deg,	R =   90.000 deg
};
P[1842]{
   GP1:
	UF : 0, UT : 6,		CONFIG : 'N U T, 0, 0, 0',
	X =  46.958  mm,	Y =   -256.416  mm,	Z =   -257.344  mm,
	W =  90.000 deg,	P =   0.000 deg,	R =   90.000 deg
};
P[1843]{
   GP1:
	UF : 0, UT : 6,		CONFIG : 'N U T, 0, 0, 0',
	X =  42.744  mm,	Y =   -258.759  mm,	Z =   -257.123  mm,
	W =  90.000 deg,	P =   0.000 deg,	R =   90.000 deg
};
P[1844]{
   GP1:
	UF : 0, UT : 6,		CONFIG : 'N U T, 0, 0, 0',
	X =  41.741  mm,	Y =   -259.338  mm,	Z =   -257.123  mm,
	W =  90.000 deg,	P =   0.000 deg,	R =   90.000 deg
};
P[1845]{
   GP1:
	UF : 0, UT : 6,		CONFIG : 'N U T, 0, 0, 0',
	X =  35.191  mm,	Y =   -263.113  mm,	Z =   -257.107  mm,
	W =  90.000 deg,	P =   0.000 deg,	R =   90.000 deg
};
P[1846]{
   GP1:
	UF : 0, UT : 6,		CONFIG : 'N U T, 0, 0, 0',
	X =  34.352  mm,	Y =   -263.613  mm,	Z =   -257.146  mm,
	W =  90.000 deg,	P =   0.000 deg,	R =   90.000 deg
};
P[1847]{
   GP1:
	UF : 0, UT : 6,		CONFIG : 'N U T, 0, 0, 0',
	X =  23.205  mm,	Y =   -269.977  mm,	Z =   -256.971  mm,
	W =  90.000 deg,	P =   0.000 deg,	R =   90.000 deg
};
P[1848]{
   GP1:
	UF : 0, UT : 6,		CONFIG : 'N U T, 0, 0, 0',
	X =  20.825  mm,	Y =   -271.493  mm,	Z =   -257.314  mm,
	W =  90.000 deg,	P =   0.000 deg,	R =   90.000 deg
};
P[1849]{
   GP1:
	UF : 0, UT : 6,		CONFIG : 'N U T, 0, 0, 0',
	X =  17.381  mm,	Y =   -273.489  mm,	Z =   -257.332  mm,
	W =  90.000 deg,	P =   0.000 deg,	R =   90.000 deg
};
P[1850]{
   GP1:
	UF : 0, UT : 6,		CONFIG : 'N U T, 0, 0, 0',
	X =  16.457  mm,	Y =   -273.861  mm,	Z =   -256.940  mm,
	W =  90.000 deg,	P =   0.000 deg,	R =   90.000 deg
};
P[1851]{
   GP1:
	UF : 0, UT : 6,		CONFIG : 'N U T, 0, 0, 0',
	X =  15.645  mm,	Y =   -274.409  mm,	Z =   -257.131  mm,
	W =  90.000 deg,	P =   0.000 deg,	R =   90.000 deg
};
P[1852]{
   GP1:
	UF : 0, UT : 6,		CONFIG : 'N U T, 0, 0, 0',
	X =  14.961  mm,	Y =   -274.903  mm,	Z =   -257.373  mm,
	W =  90.000 deg,	P =   0.000 deg,	R =   90.000 deg
};
P[1853]{
   GP1:
	UF : 0, UT : 6,		CONFIG : 'N U T, 0, 0, 0',
	X =  12.129  mm,	Y =   -276.382  mm,	Z =   -256.993  mm,
	W =  90.000 deg,	P =   0.000 deg,	R =   90.000 deg
};
P[1854]{
   GP1:
	UF : 0, UT : 6,		CONFIG : 'N U T, 0, 0, 0',
	X =  11.369  mm,	Y =   -276.920  mm,	Z =   -257.234  mm,
	W =  90.000 deg,	P =   0.000 deg,	R =   90.000 deg
};
P[1855]{
   GP1:
	UF : 0, UT : 6,		CONFIG : 'N U T, 0, 0, 0',
	X =  9.106  mm,	Y =   -278.248  mm,	Z =   -257.284  mm,
	W =  90.000 deg,	P =   0.000 deg,	R =   90.000 deg
};
P[1856]{
   GP1:
	UF : 0, UT : 6,		CONFIG : 'N U T, 0, 0, 0',
	X =  0.418  mm,	Y =   -283.147  mm,	Z =   -257.000  mm,
	W =  90.000 deg,	P =   0.000 deg,	R =   90.000 deg
};
P[1857]{
   GP1:
	UF : 0, UT : 6,		CONFIG : 'N U T, 0, 0, 0',
	X =  -1.008  mm,	Y =   -284.062  mm,	Z =   -257.226  mm,
	W =  90.000 deg,	P =   0.000 deg,	R =   90.000 deg
};
P[1858]{
   GP1:
	UF : 0, UT : 6,		CONFIG : 'N U T, 0, 0, 0',
	X =  -3.600  mm,	Y =   -285.606  mm,	Z =   -257.341  mm,
	W =  90.000 deg,	P =   0.000 deg,	R =   90.000 deg
};
P[1859]{
   GP1:
	UF : 0, UT : 6,		CONFIG : 'N U T, 0, 0, 0',
	X =  -6.539  mm,	Y =   -287.169  mm,	Z =   -257.014  mm,
	W =  90.000 deg,	P =   0.000 deg,	R =   90.000 deg
};
P[1860]{
   GP1:
	UF : 0, UT : 6,		CONFIG : 'N U T, 0, 0, 0',
	X =  -10.350  mm,	Y =   -289.487  mm,	Z =   -257.299  mm,
	W =  90.000 deg,	P =   0.000 deg,	R =   90.000 deg
};
P[1861]{
   GP1:
	UF : 0, UT : 6,		CONFIG : 'N U T, 0, 0, 0',
	X =  -12.281  mm,	Y =   -290.637  mm,	Z =   -257.385  mm,
	W =  90.000 deg,	P =   0.000 deg,	R =   90.000 deg
};
P[1862]{
   GP1:
	UF : 0, UT : 6,		CONFIG : 'N U T, 0, 0, 0',
	X =  -13.898  mm,	Y =   -291.407  mm,	Z =   -256.986  mm,
	W =  90.000 deg,	P =   0.000 deg,	R =   90.000 deg
};
P[1863]{
   GP1:
	UF : 0, UT : 6,		CONFIG : 'N U T, 0, 0, 0',
	X =  -14.668  mm,	Y =   -292.001  mm,	Z =   -257.349  mm,
	W =  90.000 deg,	P =   0.000 deg,	R =   90.000 deg
};
P[1864]{
   GP1:
	UF : 0, UT : 6,		CONFIG : 'N U T, 0, 0, 0',
	X =  -15.744  mm,	Y =   -292.489  mm,	Z =   -257.027  mm,
	W =  90.000 deg,	P =   0.000 deg,	R =   90.000 deg
};
P[1865]{
   GP1:
	UF : 0, UT : 6,		CONFIG : 'N U T, 0, 0, 0',
	X =  -16.379  mm,	Y =   -292.918  mm,	Z =   -257.177  mm,
	W =  90.000 deg,	P =   0.000 deg,	R =   90.000 deg
};
P[1866]{
   GP1:
	UF : 0, UT : 6,		CONFIG : 'N U T, 0, 0, 0',
	X =  -19.853  mm,	Y =   -294.965  mm,	Z =   -257.279  mm,
	W =  90.000 deg,	P =   0.000 deg,	R =   90.000 deg
};
P[1867]{
   GP1:
	UF : 0, UT : 6,		CONFIG : 'N U T, 0, 0, 0',
	X =  -22.787  mm,	Y =   -296.547  mm,	Z =   -257.006  mm,
	W =  90.000 deg,	P =   0.000 deg,	R =   90.000 deg
};
P[1868]{
   GP1:
	UF : 0, UT : 6,		CONFIG : 'N U T, 0, 0, 0',
	X =  -23.247  mm,	Y =   -296.925  mm,	Z =   -257.276  mm,
	W =  90.000 deg,	P =   0.000 deg,	R =   90.000 deg
};
P[1869]{
   GP1:
	UF : 0, UT : 6,		CONFIG : 'N U T, 0, 0, 0',
	X =  -27.498  mm,	Y =   -299.400  mm,	Z =   -257.328  mm,
	W =  90.000 deg,	P =   0.000 deg,	R =   90.000 deg
};
P[1870]{
   GP1:
	UF : 0, UT : 6,		CONFIG : 'N U T, 0, 0, 0',
	X =  -28.122  mm,	Y =   -299.638  mm,	Z =   -257.031  mm,
	W =  90.000 deg,	P =   0.000 deg,	R =   90.000 deg
};
P[1871]{
   GP1:
	UF : 0, UT : 6,		CONFIG : 'N U T, 0, 0, 0',
	X =  -29.230  mm,	Y =   -300.226  mm,	Z =   -256.908  mm,
	W =  90.000 deg,	P =   0.000 deg,	R =   90.000 deg
};
P[1872]{
   GP1:
	UF : 0, UT : 6,		CONFIG : 'N U T, 0, 0, 0',
	X =  -29.807  mm,	Y =   -300.610  mm,	Z =   -257.029  mm,
	W =  90.000 deg,	P =   0.000 deg,	R =   90.000 deg
};
P[1873]{
   GP1:
	UF : 0, UT : 6,		CONFIG : 'N U T, 0, 0, 0',
	X =  -30.956  mm,	Y =   -301.388  mm,	Z =   -257.307  mm,
	W =  90.000 deg,	P =   0.000 deg,	R =   90.000 deg
};
P[1874]{
   GP1:
	UF : 0, UT : 6,		CONFIG : 'N U T, 0, 0, 0',
	X =  -34.438  mm,	Y =   -303.420  mm,	Z =   -257.361  mm,
	W =  90.000 deg,	P =   0.000 deg,	R =   90.000 deg
};
P[1875]{
   GP1:
	UF : 0, UT : 6,		CONFIG : 'N U T, 0, 0, 0',
	X =  -36.548  mm,	Y =   -304.599  mm,	Z =   -257.263  mm,
	W =  90.000 deg,	P =   0.000 deg,	R =   90.000 deg
};
P[1876]{
   GP1:
	UF : 0, UT : 6,		CONFIG : 'N U T, 0, 0, 0',
	X =  -40.904  mm,	Y =   -307.045  mm,	Z =   -257.096  mm,
	W =  90.000 deg,	P =   0.000 deg,	R =   90.000 deg
};
P[1877]{
   GP1:
	UF : 0, UT : 6,		CONFIG : 'N U T, 0, 0, 0',
	X =  -42.598  mm,	Y =   -308.025  mm,	Z =   -257.102  mm,
	W =  90.000 deg,	P =   0.000 deg,	R =   90.000 deg
};
P[1878]{
   GP1:
	UF : 0, UT : 6,		CONFIG : 'N U T, 0, 0, 0',
	X =  -45.027  mm,	Y =   -309.449  mm,	Z =   -257.155  mm,
	W =  90.000 deg,	P =   0.000 deg,	R =   90.000 deg
};
P[1879]{
   GP1:
	UF : 0, UT : 6,		CONFIG : 'N U T, 0, 0, 0',
	X =  -45.814  mm,	Y =   -309.928  mm,	Z =   -257.215  mm,
	W =  90.000 deg,	P =   0.000 deg,	R =   90.000 deg
};
P[1880]{
   GP1:
	UF : 0, UT : 6,		CONFIG : 'N U T, 0, 0, 0',
	X =  -47.757  mm,	Y =   -311.061  mm,	Z =   -257.239  mm,
	W =  90.000 deg,	P =   0.000 deg,	R =   90.000 deg
};
P[1881]{
   GP1:
	UF : 0, UT : 6,		CONFIG : 'N U T, 0, 0, 0',
	X =  -50.492  mm,	Y =   -312.568  mm,	Z =   -257.063  mm,
	W =  90.000 deg,	P =   0.000 deg,	R =   90.000 deg
};
P[1882]{
   GP1:
	UF : 0, UT : 6,		CONFIG : 'N U T, 0, 0, 0',
	X =  -51.970  mm,	Y =   -313.400  mm,	Z =   -257.012  mm,
	W =  90.000 deg,	P =   0.000 deg,	R =   90.000 deg
};
P[1883]{
   GP1:
	UF : 0, UT : 6,		CONFIG : 'N U T, 0, 0, 0',
	X =  -53.647  mm,	Y =   -314.452  mm,	Z =   -257.216  mm,
	W =  90.000 deg,	P =   0.000 deg,	R =   90.000 deg
};
P[1884]{
   GP1:
	UF : 0, UT : 6,		CONFIG : 'N U T, 0, 0, 0',
	X =  -54.611  mm,	Y =   -314.944  mm,	Z =   -257.061  mm,
	W =  90.000 deg,	P =   0.000 deg,	R =   90.000 deg
};
P[1885]{
   GP1:
	UF : 0, UT : 6,		CONFIG : 'N U T, 0, 0, 0',
	X =  -57.352  mm,	Y =   -316.597  mm,	Z =   -257.228  mm,
	W =  90.000 deg,	P =   0.000 deg,	R =   90.000 deg
};
P[1886]{
   GP1:
	UF : 0, UT : 6,		CONFIG : 'N U T, 0, 0, 0',
	X =  -61.561  mm,	Y =   -319.017  mm,	Z =   -257.205  mm,
	W =  90.000 deg,	P =   0.000 deg,	R =   90.000 deg
};
P[1887]{
   GP1:
	UF : 0, UT : 6,		CONFIG : 'N U T, 0, 0, 0',
	X =  -62.161  mm,	Y =   -319.352  mm,	Z =   -257.174  mm,
	W =  90.000 deg,	P =   0.000 deg,	R =   90.000 deg
};
P[1888]{
   GP1:
	UF : 0, UT : 6,		CONFIG : 'N U T, 0, 0, 0',
	X =  -66.003  mm,	Y =   -321.656  mm,	Z =   -257.383  mm,
	W =  90.000 deg,	P =   0.000 deg,	R =   90.000 deg
};
P[1889]{
   GP1:
	UF : 0, UT : 6,		CONFIG : 'N U T, 0, 0, 0',
	X =  -68.128  mm,	Y =   -322.834  mm,	Z =   -257.266  mm,
	W =  90.000 deg,	P =   0.000 deg,	R =   90.000 deg
};
P[1890]{
   GP1:
	UF : 0, UT : 6,		CONFIG : 'N U T, 0, 0, 0',
	X =  -71.437  mm,	Y =   -324.615  mm,	Z =   -256.955  mm,
	W =  90.000 deg,	P =   0.000 deg,	R =   90.000 deg
};
P[1891]{
   GP1:
	UF : 0, UT : 6,		CONFIG : 'N U T, 0, 0, 0',
	X =  -72.174  mm,	Y =   -325.061  mm,	Z =   -257.004  mm,
	W =  90.000 deg,	P =   0.000 deg,	R =   90.000 deg
};
P[1892]{
   GP1:
	UF : 0, UT : 6,		CONFIG : 'N U T, 0, 0, 0',
	X =  -75.784  mm,	Y =   -327.214  mm,	Z =   -257.167  mm,
	W =  90.000 deg,	P =   0.000 deg,	R =   90.000 deg
};
P[1893]{
   GP1:
	UF : 0, UT : 6,		CONFIG : 'N U T, 0, 0, 0',
	X =  -76.770  mm,	Y =   -327.722  mm,	Z =   -257.021  mm,
	W =  90.000 deg,	P =   0.000 deg,	R =   90.000 deg
};
P[1894]{
   GP1:
	UF : 0, UT : 6,		CONFIG : 'N U T, 0, 0, 0',
	X =  -78.342  mm,	Y =   -328.752  mm,	Z =   -257.316  mm,
	W =  90.000 deg,	P =   0.000 deg,	R =   90.000 deg
};
P[1895]{
   GP1:
	UF : 0, UT : 6,		CONFIG : 'N U T, 0, 0, 0',
	X =  -79.228  mm,	Y =   -329.190  mm,	Z =   -257.139  mm,
	W =  90.000 deg,	P =   0.000 deg,	R =   90.000 deg
};
P[1896]{
   GP1:
	UF : 0, UT : 6,		CONFIG : 'N U T, 0, 0, 0',
	X =  -80.860  mm,	Y =   -330.165  mm,	Z =   -257.216  mm,
	W =  90.000 deg,	P =   0.000 deg,	R =   90.000 deg
};
P[1897]{
   GP1:
	UF : 0, UT : 6,		CONFIG : 'N U T, 0, 0, 0',
	X =  -82.501  mm,	Y =   -331.090  mm,	Z =   -257.161  mm,
	W =  90.000 deg,	P =   0.000 deg,	R =   90.000 deg
};
P[1898]{
   GP1:
	UF : 0, UT : 6,		CONFIG : 'N U T, 0, 0, 0',
	X =  -83.358  mm,	Y =   -331.626  mm,	Z =   -257.264  mm,
	W =  90.000 deg,	P =   0.000 deg,	R =   90.000 deg
};
P[1899]{
   GP1:
	UF : 0, UT : 6,		CONFIG : 'N U T, 0, 0, 0',
	X =  -85.833  mm,	Y =   -333.014  mm,	Z =   -257.162  mm,
	W =  90.000 deg,	P =   0.000 deg,	R =   90.000 deg
};
P[1900]{
   GP1:
	UF : 0, UT : 6,		CONFIG : 'N U T, 0, 0, 0',
	X =  -86.773  mm,	Y =   -333.546  mm,	Z =   -257.137  mm,
	W =  90.000 deg,	P =   0.000 deg,	R =   90.000 deg
};
P[1901]{
   GP1:
	UF : 0, UT : 6,		CONFIG : 'N U T, 0, 0, 0',
	X =  -88.649  mm,	Y =   -334.684  mm,	Z =   -257.269  mm,
	W =  90.000 deg,	P =   0.000 deg,	R =   90.000 deg
};
P[1902]{
   GP1:
	UF : 0, UT : 6,		CONFIG : 'N U T, 0, 0, 0',
	X =  -91.020  mm,	Y =   -335.935  mm,	Z =   -256.983  mm,
	W =  90.000 deg,	P =   0.000 deg,	R =   90.000 deg
};
P[1903]{
   GP1:
	UF : 0, UT : 6,		CONFIG : 'N U T, 0, 0, 0',
	X =  -91.783  mm,	Y =   -336.407  mm,	Z =   -257.060  mm,
	W =  90.000 deg,	P =   0.000 deg,	R =   90.000 deg
};
P[1904]{
   GP1:
	UF : 0, UT : 6,		CONFIG : 'N U T, 0, 0, 0',
	X =  -93.729  mm,	Y =   -337.660  mm,	Z =   -257.373  mm,
	W =  90.000 deg,	P =   0.000 deg,	R =   90.000 deg
};
P[1905]{
   GP1:
	UF : 0, UT : 6,		CONFIG : 'N U T, 0, 0, 0',
	X =  -94.547  mm,	Y =   -338.119  mm,	Z =   -257.341  mm,
	W =  90.000 deg,	P =   0.000 deg,	R =   90.000 deg
};
P[1906]{
   GP1:
	UF : 0, UT : 6,		CONFIG : 'N U T, 0, 0, 0',
	X =  -95.237  mm,	Y =   -338.518  mm,	Z =   -257.343  mm,
	W =  90.000 deg,	P =   0.000 deg,	R =   90.000 deg
};
P[1907]{
   GP1:
	UF : 0, UT : 6,		CONFIG : 'N U T, 0, 0, 0',
	X =  -99.668  mm,	Y =   -341.086  mm,	Z =   -257.364  mm,
	W =  90.000 deg,	P =   0.000 deg,	R =   90.000 deg
};
P[1908]{
   GP1:
	UF : 0, UT : 6,		CONFIG : 'N U T, 0, 0, 0',
	X =  -101.212  mm,	Y =   -341.798  mm,	Z =   -256.932  mm,
	W =  90.000 deg,	P =   0.000 deg,	R =   90.000 deg
};
P[1909]{
   GP1:
	UF : 0, UT : 6,		CONFIG : 'N U T, 0, 0, 0',
	X =  -102.073  mm,	Y =   -342.316  mm,	Z =   -256.982  mm,
	W =  90.000 deg,	P =   0.000 deg,	R =   90.000 deg
};
P[1910]{
   GP1:
	UF : 0, UT : 6,		CONFIG : 'N U T, 0, 0, 0',
	X =  -103.913  mm,	Y =   -343.468  mm,	Z =   -257.196  mm,
	W =  90.000 deg,	P =   0.000 deg,	R =   90.000 deg
};
P[1911]{
   GP1:
	UF : 0, UT : 6,		CONFIG : 'N U T, 0, 0, 0',
	X =  -106.499  mm,	Y =   -344.895  mm,	Z =   -257.038  mm,
	W =  90.000 deg,	P =   0.000 deg,	R =   90.000 deg
};
P[1912]{
   GP1:
	UF : 0, UT : 6,		CONFIG : 'N U T, 0, 0, 0',
	X =  -107.885  mm,	Y =   -345.831  mm,	Z =   -257.368  mm,
	W =  90.000 deg,	P =   0.000 deg,	R =   90.000 deg
};
P[1913]{
   GP1:
	UF : 0, UT : 6,		CONFIG : 'N U T, 0, 0, 0',
	X =  -109.769  mm,	Y =   -346.844  mm,	Z =   -257.186  mm,
	W =  90.000 deg,	P =   0.000 deg,	R =   90.000 deg
};
P[1914]{
   GP1:
	UF : 0, UT : 6,		CONFIG : 'N U T, 0, 0, 0',
	X =  -110.945  mm,	Y =   -347.551  mm,	Z =   -257.253  mm,
	W =  90.000 deg,	P =   0.000 deg,	R =   90.000 deg
};
P[1915]{
   GP1:
	UF : 0, UT : 6,		CONFIG : 'N U T, 0, 0, 0',
	X =  -112.551  mm,	Y =   -348.390  mm,	Z =   -257.039  mm,
	W =  90.000 deg,	P =   0.000 deg,	R =   90.000 deg
};
P[1916]{
   GP1:
	UF : 0, UT : 6,		CONFIG : 'N U T, 0, 0, 0',
	X =  -115.132  mm,	Y =   -350.023  mm,	Z =   -257.185  mm,
	W =  90.000 deg,	P =   0.000 deg,	R =   90.000 deg
};
P[1917]{
   GP1:
	UF : 0, UT : 6,		CONFIG : 'N U T, 0, 0, 0',
	X =  -116.227  mm,	Y =   -350.866  mm,	Z =   -257.303  mm,
	W =  90.000 deg,	P =   0.000 deg,	R =   90.000 deg
};
P[1918]{
   GP1:
	UF : 0, UT : 6,		CONFIG : 'N U T, 0, 0, 0',
	X =  -117.088  mm,	Y =   -351.525  mm,	Z =   -257.239  mm,
	W =  90.000 deg,	P =   0.000 deg,	R =   90.000 deg
};
P[1919]{
   GP1:
	UF : 0, UT : 6,		CONFIG : 'N U T, 0, 0, 0',
	X =  -118.466  mm,	Y =   -353.038  mm,	Z =   -257.271  mm,
	W =  90.000 deg,	P =   0.000 deg,	R =   90.000 deg
};
P[1920]{
   GP1:
	UF : 0, UT : 6,		CONFIG : 'N U T, 0, 0, 0',
	X =  -119.348  mm,	Y =   -353.919  mm,	Z =   -256.887  mm,
	W =  90.000 deg,	P =   0.000 deg,	R =   90.000 deg
};
P[1921]{
   GP1:
	UF : 0, UT : 6,		CONFIG : 'N U T, 0, 0, 0',
	X =  -120.411  mm,	Y =   -356.196  mm,	Z =   -257.232  mm,
	W =  90.000 deg,	P =   0.000 deg,	R =   90.000 deg
};
P[1922]{
   GP1:
	UF : 0, UT : 6,		CONFIG : 'N U T, 0, 0, 0',
	X =  -121.326  mm,	Y =   -359.925  mm,	Z =   -257.365  mm,
	W =  90.000 deg,	P =   0.000 deg,	R =   90.000 deg
};
P[1923]{
   GP1:
	UF : 0, UT : 6,		CONFIG : 'N U T, 0, 0, 0',
	X =  -121.247  mm,	Y =   -363.620  mm,	Z =   -257.249  mm,
	W =  90.000 deg,	P =   0.000 deg,	R =   90.000 deg
};
P[1924]{
   GP1:
	UF : 0, UT : 6,		CONFIG : 'N U T, 0, 0, 0',
	X =  -120.816  mm,	Y =   -365.863  mm,	Z =   -257.002  mm,
	W =  90.000 deg,	P =   0.000 deg,	R =   90.000 deg
};
P[1925]{
   GP1:
	UF : 0, UT : 6,		CONFIG : 'N U T, 0, 0, 0',
	X =  -120.266  mm,	Y =   -366.987  mm,	Z =   -257.122  mm,
	W =  90.000 deg,	P =   0.000 deg,	R =   90.000 deg
};
P[1926]{
   GP1:
	UF : 0, UT : 6,		CONFIG : 'N U T, 0, 0, 0',
	X =  -119.300  mm,	Y =   -369.089  mm,	Z =   -256.942  mm,
	W =  90.000 deg,	P =   0.000 deg,	R =   90.000 deg
};
P[1927]{
   GP1:
	UF : 0, UT : 6,		CONFIG : 'N U T, 0, 0, 0',
	X =  -118.482  mm,	Y =   -370.279  mm,	Z =   -257.261  mm,
	W =  90.000 deg,	P =   0.000 deg,	R =   90.000 deg
};
P[1928]{
   GP1:
	UF : 0, UT : 6,		CONFIG : 'N U T, 0, 0, 0',
	X =  -116.694  mm,	Y =   -373.330  mm,	Z =   -257.324  mm,
	W =  90.000 deg,	P =   0.000 deg,	R =   90.000 deg
};
P[1929]{
   GP1:
	UF : 0, UT : 6,		CONFIG : 'N U T, 0, 0, 0',
	X =  -115.079  mm,	Y =   -376.086  mm,	Z =   -257.381  mm,
	W =  90.000 deg,	P =   0.000 deg,	R =   90.000 deg
};
P[1930]{
   GP1:
	UF : 0, UT : 6,		CONFIG : 'N U T, 0, 0, 0',
	X =  -113.240  mm,	Y =   -379.310  mm,	Z =   -257.326  mm,
	W =  90.000 deg,	P =   0.000 deg,	R =   90.000 deg
};
P[1931]{
   GP1:
	UF : 0, UT : 6,		CONFIG : 'N U T, 0, 0, 0',
	X =  -112.549  mm,	Y =   -380.646  mm,	Z =   -257.131  mm,
	W =  90.000 deg,	P =   0.000 deg,	R =   90.000 deg
};
P[1932]{
   GP1:
	UF : 0, UT : 6,		CONFIG : 'N U T, 0, 0, 0',
	X =  -110.189  mm,	Y =   -384.819  mm,	Z =   -257.012  mm,
	W =  90.000 deg,	P =   0.000 deg,	R =   90.000 deg
};
P[1933]{
   GP1:
	UF : 0, UT : 6,		CONFIG : 'N U T, 0, 0, 0',
	X =  -109.577  mm,	Y =   -385.708  mm,	Z =   -257.252  mm,
	W =  90.000 deg,	P =   0.000 deg,	R =   90.000 deg
};
P[1934]{
   GP1:
	UF : 0, UT : 6,		CONFIG : 'N U T, 0, 0, 0',
	X =  -108.832  mm,	Y =   -386.983  mm,	Z =   -257.272  mm,
	W =  90.000 deg,	P =   0.000 deg,	R =   90.000 deg
};
P[1935]{
   GP1:
	UF : 0, UT : 6,		CONFIG : 'N U T, 0, 0, 0',
	X =  -108.457  mm,	Y =   -387.727  mm,	Z =   -257.140  mm,
	W =  90.000 deg,	P =   0.000 deg,	R =   90.000 deg
};
P[1936]{
   GP1:
	UF : 0, UT : 6,		CONFIG : 'N U T, 0, 0, 0',
	X =  -108.050  mm,	Y =   -388.372  mm,	Z =   -257.224  mm,
	W =  90.000 deg,	P =   0.000 deg,	R =   90.000 deg
};
P[1937]{
   GP1:
	UF : 0, UT : 6,		CONFIG : 'N U T, 0, 0, 0',
	X =  -106.937  mm,	Y =   -390.271  mm,	Z =   -257.262  mm,
	W =  90.000 deg,	P =   0.000 deg,	R =   90.000 deg
};
P[1938]{
   GP1:
	UF : 0, UT : 6,		CONFIG : 'N U T, 0, 0, 0',
	X =  -104.854  mm,	Y =   -393.799  mm,	Z =   -257.377  mm,
	W =  90.000 deg,	P =   0.000 deg,	R =   90.000 deg
};
P[1939]{
   GP1:
	UF : 0, UT : 6,		CONFIG : 'N U T, 0, 0, 0',
	X =  -103.300  mm,	Y =   -396.529  mm,	Z =   -257.320  mm,
	W =  90.000 deg,	P =   0.000 deg,	R =   90.000 deg
};
P[1940]{
   GP1:
	UF : 0, UT : 6,		CONFIG : 'N U T, 0, 0, 0',
	X =  -103.043  mm,	Y =   -397.194  mm,	Z =   -257.014  mm,
	W =  90.000 deg,	P =   0.000 deg,	R =   90.000 deg
};
P[1941]{
   GP1:
	UF : 0, UT : 6,		CONFIG : 'N U T, 0, 0, 0',
	X =  -102.513  mm,	Y =   -398.045  mm,	Z =   -257.107  mm,
	W =  90.000 deg,	P =   0.000 deg,	R =   90.000 deg
};
P[1942]{
   GP1:
	UF : 0, UT : 6,		CONFIG : 'N U T, 0, 0, 0',
	X =  -101.847  mm,	Y =   -399.179  mm,	Z =   -257.135  mm,
	W =  90.000 deg,	P =   0.000 deg,	R =   90.000 deg
};
P[1943]{
   GP1:
	UF : 0, UT : 6,		CONFIG : 'N U T, 0, 0, 0',
	X =  -100.505  mm,	Y =   -401.472  mm,	Z =   -257.178  mm,
	W =  90.000 deg,	P =   0.000 deg,	R =   90.000 deg
};
P[1944]{
   GP1:
	UF : 0, UT : 6,		CONFIG : 'N U T, 0, 0, 0',
	X =  -99.446  mm,	Y =   -403.381  mm,	Z =   -257.071  mm,
	W =  90.000 deg,	P =   0.000 deg,	R =   90.000 deg
};
P[1945]{
   GP1:
	UF : 0, UT : 6,		CONFIG : 'N U T, 0, 0, 0',
	X =  -98.710  mm,	Y =   -404.575  mm,	Z =   -257.187  mm,
	W =  90.000 deg,	P =   0.000 deg,	R =   90.000 deg
};
P[1946]{
   GP1:
	UF : 0, UT : 6,		CONFIG : 'N U T, 0, 0, 0',
	X =  -98.046  mm,	Y =   -405.704  mm,	Z =   -257.213  mm,
	W =  90.000 deg,	P =   0.000 deg,	R =   90.000 deg
};
P[1947]{
   GP1:
	UF : 0, UT : 6,		CONFIG : 'N U T, 0, 0, 0',
	X =  -97.208  mm,	Y =   -407.253  mm,	Z =   -257.080  mm,
	W =  90.000 deg,	P =   0.000 deg,	R =   90.000 deg
};
P[1948]{
   GP1:
	UF : 0, UT : 6,		CONFIG : 'N U T, 0, 0, 0',
	X =  -93.792  mm,	Y =   -413.162  mm,	Z =   -257.089  mm,
	W =  90.000 deg,	P =   0.000 deg,	R =   90.000 deg
};
P[1949]{
   GP1:
	UF : 0, UT : 6,		CONFIG : 'N U T, 0, 0, 0',
	X =  -92.043  mm,	Y =   -415.985  mm,	Z =   -257.378  mm,
	W =  90.000 deg,	P =   0.000 deg,	R =   90.000 deg
};
P[1950]{
   GP1:
	UF : 0, UT : 6,		CONFIG : 'N U T, 0, 0, 0',
	X =  -90.691  mm,	Y =   -418.415  mm,	Z =   -257.254  mm,
	W =  90.000 deg,	P =   0.000 deg,	R =   90.000 deg
};
P[1951]{
   GP1:
	UF : 0, UT : 6,		CONFIG : 'N U T, 0, 0, 0',
	X =  -89.183  mm,	Y =   -420.979  mm,	Z =   -257.321  mm,
	W =  90.000 deg,	P =   0.000 deg,	R =   90.000 deg
};
P[1952]{
   GP1:
	UF : 0, UT : 6,		CONFIG : 'N U T, 0, 0, 0',
	X =  -87.431  mm,	Y =   -424.271  mm,	Z =   -256.960  mm,
	W =  90.000 deg,	P =   0.000 deg,	R =   90.000 deg
};
P[1953]{
   GP1:
	UF : 0, UT : 6,		CONFIG : 'N U T, 0, 0, 0',
	X =  -85.015  mm,	Y =   -428.183  mm,	Z =   -257.340  mm,
	W =  90.000 deg,	P =   0.000 deg,	R =   90.000 deg
};
P[1954]{
   GP1:
	UF : 0, UT : 6,		CONFIG : 'N U T, 0, 0, 0',
	X =  -83.421  mm,	Y =   -430.947  mm,	Z =   -257.336  mm,
	W =  90.000 deg,	P =   0.000 deg,	R =   90.000 deg
};
P[1955]{
   GP1:
	UF : 0, UT : 6,		CONFIG : 'N U T, 0, 0, 0',
	X =  -82.380  mm,	Y =   -432.760  mm,	Z =   -257.321  mm,
	W =  90.000 deg,	P =   0.000 deg,	R =   90.000 deg
};
P[1956]{
   GP1:
	UF : 0, UT : 6,		CONFIG : 'N U T, 0, 0, 0',
	X =  -81.175  mm,	Y =   -435.032  mm,	Z =   -257.063  mm,
	W =  90.000 deg,	P =   0.000 deg,	R =   90.000 deg
};
P[1957]{
   GP1:
	UF : 0, UT : 6,		CONFIG : 'N U T, 0, 0, 0',
	X =  -79.979  mm,	Y =   -436.893  mm,	Z =   -257.357  mm,
	W =  90.000 deg,	P =   0.000 deg,	R =   90.000 deg
};
P[1958]{
   GP1:
	UF : 0, UT : 6,		CONFIG : 'N U T, 0, 0, 0',
	X =  -77.649  mm,	Y =   -440.994  mm,	Z =   -257.267  mm,
	W =  90.000 deg,	P =   0.000 deg,	R =   90.000 deg
};
P[1959]{
   GP1:
	UF : 0, UT : 6,		CONFIG : 'N U T, 0, 0, 0',
	X =  -76.948  mm,	Y =   -442.135  mm,	Z =   -257.366  mm,
	W =  90.000 deg,	P =   0.000 deg,	R =   90.000 deg
};
P[1960]{
   GP1:
	UF : 0, UT : 6,		CONFIG : 'N U T, 0, 0, 0',
	X =  -76.530  mm,	Y =   -443.071  mm,	Z =   -257.070  mm,
	W =  90.000 deg,	P =   0.000 deg,	R =   90.000 deg
};
P[1961]{
   GP1:
	UF : 0, UT : 6,		CONFIG : 'N U T, 0, 0, 0',
	X =  -75.644  mm,	Y =   -444.703  mm,	Z =   -256.933  mm,
	W =  90.000 deg,	P =   0.000 deg,	R =   90.000 deg
};
P[1962]{
   GP1:
	UF : 0, UT : 6,		CONFIG : 'N U T, 0, 0, 0',
	X =  -74.633  mm,	Y =   -446.183  mm,	Z =   -257.314  mm,
	W =  90.000 deg,	P =   0.000 deg,	R =   90.000 deg
};
P[1963]{
   GP1:
	UF : 0, UT : 6,		CONFIG : 'N U T, 0, 0, 0',
	X =  -74.254  mm,	Y =   -446.875  mm,	Z =   -257.265  mm,
	W =  90.000 deg,	P =   0.000 deg,	R =   90.000 deg
};
P[1964]{
   GP1:
	UF : 0, UT : 6,		CONFIG : 'N U T, 0, 0, 0',
	X =  -73.286  mm,	Y =   -448.574  mm,	Z =   -257.233  mm,
	W =  90.000 deg,	P =   0.000 deg,	R =   90.000 deg
};
P[1965]{
   GP1:
	UF : 0, UT : 6,		CONFIG : 'N U T, 0, 0, 0',
	X =  -72.458  mm,	Y =   -450.013  mm,	Z =   -257.226  mm,
	W =  90.000 deg,	P =   0.000 deg,	R =   90.000 deg
};
P[1966]{
   GP1:
	UF : 0, UT : 6,		CONFIG : 'N U T, 0, 0, 0',
	X =  -69.387  mm,	Y =   -455.325  mm,	Z =   -257.235  mm,
	W =  90.000 deg,	P =   0.000 deg,	R =   90.000 deg
};
P[1967]{
   GP1:
	UF : 0, UT : 6,		CONFIG : 'N U T, 0, 0, 0',
	X =  -68.903  mm,	Y =   -456.409  mm,	Z =   -256.890  mm,
	W =  90.000 deg,	P =   0.000 deg,	R =   90.000 deg
};
P[1968]{
   GP1:
	UF : 0, UT : 6,		CONFIG : 'N U T, 0, 0, 0',
	X =  -68.327  mm,	Y =   -457.157  mm,	Z =   -257.242  mm,
	W =  90.000 deg,	P =   0.000 deg,	R =   90.000 deg
};
P[1969]{
   GP1:
	UF : 0, UT : 6,		CONFIG : 'N U T, 0, 0, 0',
	X =  -67.317  mm,	Y =   -458.895  mm,	Z =   -257.258  mm,
	W =  90.000 deg,	P =   0.000 deg,	R =   90.000 deg
};
P[1970]{
   GP1:
	UF : 0, UT : 6,		CONFIG : 'N U T, 0, 0, 0',
	X =  -66.466  mm,	Y =   -460.493  mm,	Z =   -257.083  mm,
	W =  90.000 deg,	P =   0.000 deg,	R =   90.000 deg
};
P[1971]{
   GP1:
	UF : 0, UT : 6,		CONFIG : 'N U T, 0, 0, 0',
	X =  -65.816  mm,	Y =   -461.558  mm,	Z =   -257.166  mm,
	W =  90.000 deg,	P =   0.000 deg,	R =   90.000 deg
};
P[1972]{
   GP1:
	UF : 0, UT : 6,		CONFIG : 'N U T, 0, 0, 0',
	X =  -65.431  mm,	Y =   -462.119  mm,	Z =   -257.316  mm,
	W =  90.000 deg,	P =   0.000 deg,	R =   90.000 deg
};
P[1973]{
   GP1:
	UF : 0, UT : 6,		CONFIG : 'N U T, 0, 0, 0',
	X =  -63.677  mm,	Y =   -465.249  mm,	Z =   -257.187  mm,
	W =  90.000 deg,	P =   0.000 deg,	R =   90.000 deg
};
P[1974]{
   GP1:
	UF : 0, UT : 6,		CONFIG : 'N U T, 0, 0, 0',
	X =  -62.883  mm,	Y =   -466.594  mm,	Z =   -257.229  mm,
	W =  90.000 deg,	P =   0.000 deg,	R =   90.000 deg
};
P[1975]{
   GP1:
	UF : 0, UT : 6,		CONFIG : 'N U T, 0, 0, 0',
	X =  -62.409  mm,	Y =   -467.426  mm,	Z =   -257.215  mm,
	W =  90.000 deg,	P =   0.000 deg,	R =   90.000 deg
};
P[1976]{
   GP1:
	UF : 0, UT : 6,		CONFIG : 'N U T, 0, 0, 0',
	X =  -61.863  mm,	Y =   -468.370  mm,	Z =   -257.217  mm,
	W =  90.000 deg,	P =   0.000 deg,	R =   90.000 deg
};
P[1977]{
   GP1:
	UF : 0, UT : 6,		CONFIG : 'N U T, 0, 0, 0',
	X =  -61.103  mm,	Y =   -469.693  mm,	Z =   -257.207  mm,
	W =  90.000 deg,	P =   0.000 deg,	R =   90.000 deg
};
P[1978]{
   GP1:
	UF : 0, UT : 6,		CONFIG : 'N U T, 0, 0, 0',
	X =  -59.627  mm,	Y =   -472.170  mm,	Z =   -257.317  mm,
	W =  90.000 deg,	P =   0.000 deg,	R =   90.000 deg
};
P[1979]{
   GP1:
	UF : 0, UT : 6,		CONFIG : 'N U T, 0, 0, 0',
	X =  -58.285  mm,	Y =   -474.802  mm,	Z =   -256.887  mm,
	W =  90.000 deg,	P =   0.000 deg,	R =   90.000 deg
};
P[1980]{
   GP1:
	UF : 0, UT : 6,		CONFIG : 'N U T, 0, 0, 0',
	X =  -57.685  mm,	Y =   -475.745  mm,	Z =   -257.022  mm,
	W =  90.000 deg,	P =   0.000 deg,	R =   90.000 deg
};
P[1981]{
   GP1:
	UF : 0, UT : 6,		CONFIG : 'N U T, 0, 0, 0',
	X =  -56.787  mm,	Y =   -477.090  mm,	Z =   -257.315  mm,
	W =  90.000 deg,	P =   0.000 deg,	R =   90.000 deg
};
P[1982]{
   GP1:
	UF : 0, UT : 6,		CONFIG : 'N U T, 0, 0, 0',
	X =  -56.170  mm,	Y =   -478.458  mm,	Z =   -256.896  mm,
	W =  90.000 deg,	P =   0.000 deg,	R =   90.000 deg
};
P[1983]{
   GP1:
	UF : 0, UT : 6,		CONFIG : 'N U T, 0, 0, 0',
	X =  -55.124  mm,	Y =   -480.227  mm,	Z =   -256.956  mm,
	W =  90.000 deg,	P =   0.000 deg,	R =   90.000 deg
};
P[1984]{
   GP1:
	UF : 0, UT : 6,		CONFIG : 'N U T, 0, 0, 0',
	X =  -54.550  mm,	Y =   -480.988  mm,	Z =   -257.282  mm,
	W =  90.000 deg,	P =   0.000 deg,	R =   90.000 deg
};
P[1985]{
   GP1:
	UF : 0, UT : 6,		CONFIG : 'N U T, 0, 0, 0',
	X =  -51.961  mm,	Y =   -485.444  mm,	Z =   -257.322  mm,
	W =  90.000 deg,	P =   0.000 deg,	R =   90.000 deg
};
P[1986]{
   GP1:
	UF : 0, UT : 6,		CONFIG : 'N U T, 0, 0, 0',
	X =  -51.672  mm,	Y =   -486.053  mm,	Z =   -257.171  mm,
	W =  90.000 deg,	P =   0.000 deg,	R =   90.000 deg
};
P[1987]{
   GP1:
	UF : 0, UT : 6,		CONFIG : 'N U T, 0, 0, 0',
	X =  -51.153  mm,	Y =   -487.027  mm,	Z =   -257.065  mm,
	W =  90.000 deg,	P =   0.000 deg,	R =   90.000 deg
};
P[1988]{
   GP1:
	UF : 0, UT : 6,		CONFIG : 'N U T, 0, 0, 0',
	X =  -50.653  mm,	Y =   -487.855  mm,	Z =   -257.118  mm,
	W =  90.000 deg,	P =   0.000 deg,	R =   90.000 deg
};
P[1989]{
   GP1:
	UF : 0, UT : 6,		CONFIG : 'N U T, 0, 0, 0',
	X =  -49.107  mm,	Y =   -490.415  mm,	Z =   -257.284  mm,
	W =  90.000 deg,	P =   0.000 deg,	R =   90.000 deg
};
P[1990]{
   GP1:
	UF : 0, UT : 6,		CONFIG : 'N U T, 0, 0, 0',
	X =  -48.122  mm,	Y =   -492.064  mm,	Z =   -257.361  mm,
	W =  90.000 deg,	P =   0.000 deg,	R =   90.000 deg
};
P[1991]{
   GP1:
	UF : 0, UT : 6,		CONFIG : 'N U T, 0, 0, 0',
	X =  -47.195  mm,	Y =   -493.909  mm,	Z =   -257.026  mm,
	W =  90.000 deg,	P =   0.000 deg,	R =   90.000 deg
};
P[1992]{
   GP1:
	UF : 0, UT : 6,		CONFIG : 'N U T, 0, 0, 0',
	X =  -46.241  mm,	Y =   -495.341  mm,	Z =   -257.337  mm,
	W =  90.000 deg,	P =   0.000 deg,	R =   90.000 deg
};
P[1993]{
   GP1:
	UF : 0, UT : 6,		CONFIG : 'N U T, 0, 0, 0',
	X =  -45.753  mm,	Y =   -496.181  mm,	Z =   -257.343  mm,
	W =  90.000 deg,	P =   0.000 deg,	R =   90.000 deg
};
P[1994]{
   GP1:
	UF : 0, UT : 6,		CONFIG : 'N U T, 0, 0, 0',
	X =  -44.427  mm,	Y =   -498.487  mm,	Z =   -257.329  mm,
	W =  90.000 deg,	P =   0.000 deg,	R =   90.000 deg
};
P[1995]{
   GP1:
	UF : 0, UT : 6,		CONFIG : 'N U T, 0, 0, 0',
	X =  -44.089  mm,	Y =   -499.262  mm,	Z =   -257.065  mm,
	W =  90.000 deg,	P =   0.000 deg,	R =   90.000 deg
};
P[1996]{
   GP1:
	UF : 0, UT : 6,		CONFIG : 'N U T, 0, 0, 0',
	X =  -43.195  mm,	Y =   -500.680  mm,	Z =   -257.248  mm,
	W =  90.000 deg,	P =   0.000 deg,	R =   90.000 deg
};
P[1997]{
   GP1:
	UF : 0, UT : 6,		CONFIG : 'N U T, 0, 0, 0',
	X =  -42.057  mm,	Y =   -502.887  mm,	Z =   -256.916  mm,
	W =  90.000 deg,	P =   0.000 deg,	R =   90.000 deg
};
P[1998]{
   GP1:
	UF : 0, UT : 6,		CONFIG : 'N U T, 0, 0, 0',
	X =  -41.036  mm,	Y =   -504.493  mm,	Z =   -257.143  mm,
	W =  90.000 deg,	P =   0.000 deg,	R =   90.000 deg
};
P[1999]{
   GP1:
	UF : 0, UT : 6,		CONFIG : 'N U T, 0, 0, 0',
	X =  -40.650  mm,	Y =   -505.063  mm,	Z =   -257.282  mm,
	W =  90.000 deg,	P =   0.000 deg,	R =   90.000 deg
};
P[2000]{
   GP1:
	UF : 0, UT : 6,		CONFIG : 'N U T, 0, 0, 0',
	X =  -39.758  mm,	Y =   -506.837  mm,	Z =   -256.959  mm,
	W =  90.000 deg,	P =   0.000 deg,	R =   90.000 deg
};
P[2001]{
   GP1:
	UF : 0, UT : 6,		CONFIG : 'N U T, 0, 0, 0',
	X =  -38.797  mm,	Y =   -508.504  mm,	Z =   -256.955  mm,
	W =  90.000 deg,	P =   0.000 deg,	R =   90.000 deg
};
P[2002]{
   GP1:
	UF : 0, UT : 6,		CONFIG : 'N U T, 0, 0, 0',
	X =  -37.082  mm,	Y =   -511.340  mm,	Z =   -257.144  mm,
	W =  90.000 deg,	P =   0.000 deg,	R =   90.000 deg
};
P[2003]{
   GP1:
	UF : 0, UT : 6,		CONFIG : 'N U T, 0, 0, 0',
	X =  -34.997  mm,	Y =   -515.038  mm,	Z =   -257.021  mm,
	W =  90.000 deg,	P =   0.000 deg,	R =   90.000 deg
};
P[2004]{
   GP1:
	UF : 0, UT : 6,		CONFIG : 'N U T, 0, 0, 0',
	X =  -34.606  mm,	Y =   -515.468  mm,	Z =   -257.371  mm,
	W =  90.000 deg,	P =   0.000 deg,	R =   90.000 deg
};
P[2005]{
   GP1:
	UF : 0, UT : 6,		CONFIG : 'N U T, 0, 0, 0',
	X =  -29.260  mm,	Y =   -524.844  mm,	Z =   -257.206  mm,
	W =  90.000 deg,	P =   0.000 deg,	R =   90.000 deg
};
P[2006]{
   GP1:
	UF : 0, UT : 6,		CONFIG : 'N U T, 0, 0, 0',
	X =  -28.583  mm,	Y =   -526.141  mm,	Z =   -257.029  mm,
	W =  90.000 deg,	P =   0.000 deg,	R =   90.000 deg
};
P[2007]{
   GP1:
	UF : 0, UT : 6,		CONFIG : 'N U T, 0, 0, 0',
	X =  -27.612  mm,	Y =   -527.856  mm,	Z =   -256.985  mm,
	W =  90.000 deg,	P =   0.000 deg,	R =   90.000 deg
};
P[2008]{
   GP1:
	UF : 0, UT : 6,		CONFIG : 'N U T, 0, 0, 0',
	X =  -26.121  mm,	Y =   -530.420  mm,	Z =   -257.009  mm,
	W =  90.000 deg,	P =   0.000 deg,	R =   90.000 deg
};
P[2009]{
   GP1:
	UF : 0, UT : 6,		CONFIG : 'N U T, 0, 0, 0',
	X =  -24.774  mm,	Y =   -532.562  mm,	Z =   -257.277  mm,
	W =  90.000 deg,	P =   0.000 deg,	R =   90.000 deg
};
P[2010]{
   GP1:
	UF : 0, UT : 6,		CONFIG : 'N U T, 0, 0, 0',
	X =  -23.757  mm,	Y =   -534.352  mm,	Z =   -257.236  mm,
	W =  90.000 deg,	P =   0.000 deg,	R =   90.000 deg
};
P[2011]{
   GP1:
	UF : 0, UT : 6,		CONFIG : 'N U T, 0, 0, 0',
	X =  -23.229  mm,	Y =   -535.446  mm,	Z =   -256.985  mm,
	W =  90.000 deg,	P =   0.000 deg,	R =   90.000 deg
};
P[2012]{
   GP1:
	UF : 0, UT : 6,		CONFIG : 'N U T, 0, 0, 0',
	X =  -22.769  mm,	Y =   -536.224  mm,	Z =   -257.011  mm,
	W =  90.000 deg,	P =   0.000 deg,	R =   90.000 deg
};
P[2013]{
   GP1:
	UF : 0, UT : 6,		CONFIG : 'N U T, 0, 0, 0',
	X =  -21.718  mm,	Y =   -537.837  mm,	Z =   -257.301  mm,
	W =  90.000 deg,	P =   0.000 deg,	R =   90.000 deg
};
P[2014]{
   GP1:
	UF : 0, UT : 6,		CONFIG : 'N U T, 0, 0, 0',
	X =  -20.995  mm,	Y =   -539.221  mm,	Z =   -257.119  mm,
	W =  90.000 deg,	P =   0.000 deg,	R =   90.000 deg
};
P[2015]{
   GP1:
	UF : 0, UT : 6,		CONFIG : 'N U T, 0, 0, 0',
	X =  -19.219  mm,	Y =   -542.297  mm,	Z =   -257.116  mm,
	W =  90.000 deg,	P =   0.000 deg,	R =   90.000 deg
};
P[2016]{
   GP1:
	UF : 0, UT : 6,		CONFIG : 'N U T, 0, 0, 0',
	X =  -17.556  mm,	Y =   -545.109  mm,	Z =   -257.211  mm,
	W =  90.000 deg,	P =   0.000 deg,	R =   90.000 deg
};
P[2017]{
   GP1:
	UF : 0, UT : 6,		CONFIG : 'N U T, 0, 0, 0',
	X =  -16.904  mm,	Y =   -546.149  mm,	Z =   -257.338  mm,
	W =  90.000 deg,	P =   0.000 deg,	R =   90.000 deg
};
P[2018]{
   GP1:
	UF : 0, UT : 6,		CONFIG : 'N U T, 0, 0, 0',
	X =  -14.965  mm,	Y =   -549.518  mm,	Z =   -257.322  mm,
	W =  90.000 deg,	P =   0.000 deg,	R =   90.000 deg
};
P[2019]{
   GP1:
	UF : 0, UT : 6,		CONFIG : 'N U T, 0, 0, 0',
	X =  -12.084  mm,	Y =   -554.492  mm,	Z =   -257.342  mm,
	W =  90.000 deg,	P =   0.000 deg,	R =   90.000 deg
};
P[2020]{
   GP1:
	UF : 0, UT : 6,		CONFIG : 'N U T, 0, 0, 0',
	X =  -9.081  mm,	Y =   -559.752  mm,	Z =   -257.260  mm,
	W =  90.000 deg,	P =   0.000 deg,	R =   90.000 deg
};
P[2021]{
   GP1:
	UF : 0, UT : 6,		CONFIG : 'N U T, 0, 0, 0',
	X =  -7.944  mm,	Y =   -561.761  mm,	Z =   -257.205  mm,
	W =  90.000 deg,	P =   0.000 deg,	R =   90.000 deg
};
P[2022]{
   GP1:
	UF : 0, UT : 6,		CONFIG : 'N U T, 0, 0, 0',
	X =  -5.707  mm,	Y =   -565.657  mm,	Z =   -257.176  mm,
	W =  90.000 deg,	P =   0.000 deg,	R =   90.000 deg
};
P[2023]{
   GP1:
	UF : 0, UT : 6,		CONFIG : 'N U T, 0, 0, 0',
	X =  -4.674  mm,	Y =   -567.315  mm,	Z =   -257.358  mm,
	W =  90.000 deg,	P =   0.000 deg,	R =   90.000 deg
};
P[2024]{
   GP1:
	UF : 0, UT : 6,		CONFIG : 'N U T, 0, 0, 0',
	X =  -4.432  mm,	Y =   -567.949  mm,	Z =   -257.058  mm,
	W =  90.000 deg,	P =   0.000 deg,	R =   90.000 deg
};
P[2025]{
   GP1:
	UF : 0, UT : 6,		CONFIG : 'N U T, 0, 0, 0',
	X =  -3.757  mm,	Y =   -568.924  mm,	Z =   -257.329  mm,
	W =  90.000 deg,	P =   0.000 deg,	R =   90.000 deg
};
P[2026]{
   GP1:
	UF : 0, UT : 6,		CONFIG : 'N U T, 0, 0, 0',
	X =  -2.811  mm,	Y =   -570.645  mm,	Z =   -257.216  mm,
	W =  90.000 deg,	P =   0.000 deg,	R =   90.000 deg
};
P[2027]{
   GP1:
	UF : 0, UT : 6,		CONFIG : 'N U T, 0, 0, 0',
	X =  -2.203  mm,	Y =   -571.831  mm,	Z =   -257.028  mm,
	W =  90.000 deg,	P =   0.000 deg,	R =   90.000 deg
};
P[2028]{
   GP1:
	UF : 0, UT : 6,		CONFIG : 'N U T, 0, 0, 0',
	X =  -0.610  mm,	Y =   -574.372  mm,	Z =   -257.334  mm,
	W =  90.000 deg,	P =   0.000 deg,	R =   90.000 deg
};
P[2029]{
   GP1:
	UF : 0, UT : 6,		CONFIG : 'N U T, 0, 0, 0',
	X =  -0.365  mm,	Y =   -575.026  mm,	Z =   -257.011  mm,
	W =  90.000 deg,	P =   0.000 deg,	R =   90.000 deg
};
P[2030]{
   GP1:
	UF : 0, UT : 6,		CONFIG : 'N U T, 0, 0, 0',
	X =  1.050  mm,	Y =   -577.403  mm,	Z =   -257.116  mm,
	W =  90.000 deg,	P =   0.000 deg,	R =   90.000 deg
};
P[2031]{
   GP1:
	UF : 0, UT : 6,		CONFIG : 'N U T, 0, 0, 0',
	X =  1.562  mm,	Y =   -578.124  mm,	Z =   -257.349  mm,
	W =  90.000 deg,	P =   0.000 deg,	R =   90.000 deg
};
P[2032]{
   GP1:
	UF : 0, UT : 6,		CONFIG : 'N U T, 0, 0, 0',
	X =  2.285  mm,	Y =   -579.416  mm,	Z =   -257.291  mm,
	W =  90.000 deg,	P =   0.000 deg,	R =   90.000 deg
};
P[2033]{
   GP1:
	UF : 0, UT : 6,		CONFIG : 'N U T, 0, 0, 0',
	X =  3.742  mm,	Y =   -582.089  mm,	Z =   -257.084  mm,
	W =  90.000 deg,	P =   0.000 deg,	R =   90.000 deg
};
P[2034]{
   GP1:
	UF : 0, UT : 6,		CONFIG : 'N U T, 0, 0, 0',
	X =  4.250  mm,	Y =   -582.862  mm,	Z =   -257.231  mm,
	W =  90.000 deg,	P =   0.000 deg,	R =   90.000 deg
};
P[2035]{
   GP1:
	UF : 0, UT : 6,		CONFIG : 'N U T, 0, 0, 0',
	X =  7.567  mm,	Y =   -588.665  mm,	Z =   -257.151  mm,
	W =  90.000 deg,	P =   0.000 deg,	R =   90.000 deg
};
P[2036]{
   GP1:
	UF : 0, UT : 6,		CONFIG : 'N U T, 0, 0, 0',
	X =  8.013  mm,	Y =   -589.577  mm,	Z =   -256.955  mm,
	W =  90.000 deg,	P =   0.000 deg,	R =   90.000 deg
};
P[2037]{
   GP1:
	UF : 0, UT : 6,		CONFIG : 'N U T, 0, 0, 0',
	X =  8.926  mm,	Y =   -590.854  mm,	Z =   -257.382  mm,
	W =  90.000 deg,	P =   0.000 deg,	R =   90.000 deg
};
P[2038]{
   GP1:
	UF : 0, UT : 6,		CONFIG : 'N U T, 0, 0, 0',
	X =  9.450  mm,	Y =   -591.765  mm,	Z =   -257.377  mm,
	W =  90.000 deg,	P =   0.000 deg,	R =   90.000 deg
};
P[2039]{
   GP1:
	UF : 0, UT : 6,		CONFIG : 'N U T, 0, 0, 0',
	X =  11.268  mm,	Y =   -594.936  mm,	Z =   -257.343  mm,
	W =  90.000 deg,	P =   0.000 deg,	R =   90.000 deg
};
P[2040]{
   GP1:
	UF : 0, UT : 6,		CONFIG : 'N U T, 0, 0, 0',
	X =  12.007  mm,	Y =   -596.248  mm,	Z =   -257.298  mm,
	W =  90.000 deg,	P =   0.000 deg,	R =   90.000 deg
};
P[2041]{
   GP1:
	UF : 0, UT : 6,		CONFIG : 'N U T, 0, 0, 0',
	X =  15.385  mm,	Y =   -602.197  mm,	Z =   -257.161  mm,
	W =  90.000 deg,	P =   0.000 deg,	R =   90.000 deg
};
P[2042]{
   GP1:
	UF : 0, UT : 6,		CONFIG : 'N U T, 0, 0, 0',
	X =  15.720  mm,	Y =   -602.894  mm,	Z =   -256.997  mm,
	W =  90.000 deg,	P =   0.000 deg,	R =   90.000 deg
};
P[2043]{
   GP1:
	UF : 0, UT : 6,		CONFIG : 'N U T, 0, 0, 0',
	X =  18.294  mm,	Y =   -607.130  mm,	Z =   -257.310  mm,
	W =  90.000 deg,	P =   0.000 deg,	R =   90.000 deg
};
P[2044]{
   GP1:
	UF : 0, UT : 6,		CONFIG : 'N U T, 0, 0, 0',
	X =  18.587  mm,	Y =   -607.922  mm,	Z =   -256.910  mm,
	W =  90.000 deg,	P =   0.000 deg,	R =   90.000 deg
};
P[2045]{
   GP1:
	UF : 0, UT : 6,		CONFIG : 'N U T, 0, 0, 0',
	X =  19.405  mm,	Y =   -609.015  mm,	Z =   -257.364  mm,
	W =  90.000 deg,	P =   0.000 deg,	R =   90.000 deg
};
P[2046]{
   GP1:
	UF : 0, UT : 6,		CONFIG : 'N U T, 0, 0, 0',
	X =  20.198  mm,	Y =   -610.591  mm,	Z =   -257.079  mm,
	W =  90.000 deg,	P =   0.000 deg,	R =   90.000 deg
};
P[2047]{
   GP1:
	UF : 0, UT : 6,		CONFIG : 'N U T, 0, 0, 0',
	X =  21.501  mm,	Y =   -612.766  mm,	Z =   -257.196  mm,
	W =  90.000 deg,	P =   0.000 deg,	R =   90.000 deg
};
P[2048]{
   GP1:
	UF : 0, UT : 6,		CONFIG : 'N U T, 0, 0, 0',
	X =  22.361  mm,	Y =   -614.400  mm,	Z =   -256.992  mm,
	W =  90.000 deg,	P =   0.000 deg,	R =   90.000 deg
};
P[2049]{
   GP1:
	UF : 0, UT : 6,		CONFIG : 'N U T, 0, 0, 0',
	X =  23.202  mm,	Y =   -615.581  mm,	Z =   -257.379  mm,
	W =  90.000 deg,	P =   0.000 deg,	R =   90.000 deg
};
P[2050]{
   GP1:
	UF : 0, UT : 6,		CONFIG : 'N U T, 0, 0, 0',
	X =  23.583  mm,	Y =   -616.558  mm,	Z =   -256.933  mm,
	W =  90.000 deg,	P =   0.000 deg,	R =   90.000 deg
};
P[2051]{
   GP1:
	UF : 0, UT : 6,		CONFIG : 'N U T, 0, 0, 0',
	X =  25.237  mm,	Y =   -619.201  mm,	Z =   -257.245  mm,
	W =  90.000 deg,	P =   0.000 deg,	R =   90.000 deg
};
P[2052]{
   GP1:
	UF : 0, UT : 6,		CONFIG : 'N U T, 0, 0, 0',
	X =  26.788  mm,	Y =   -621.821  mm,	Z =   -257.337  mm,
	W =  90.000 deg,	P =   0.000 deg,	R =   90.000 deg
};
P[2053]{
   GP1:
	UF : 0, UT : 6,		CONFIG : 'N U T, 0, 0, 0',
	X =  27.486  mm,	Y =   -623.185  mm,	Z =   -257.118  mm,
	W =  90.000 deg,	P =   0.000 deg,	R =   90.000 deg
};
P[2054]{
   GP1:
	UF : 0, UT : 6,		CONFIG : 'N U T, 0, 0, 0',
	X =  29.678  mm,	Y =   -626.876  mm,	Z =   -257.266  mm,
	W =  90.000 deg,	P =   0.000 deg,	R =   90.000 deg
};
P[2055]{
   GP1:
	UF : 0, UT : 6,		CONFIG : 'N U T, 0, 0, 0',
	X =  30.897  mm,	Y =   -628.911  mm,	Z =   -257.374  mm,
	W =  90.000 deg,	P =   0.000 deg,	R =   90.000 deg
};
P[2056]{
   GP1:
	UF : 0, UT : 6,		CONFIG : 'N U T, 0, 0, 0',
	X =  31.987  mm,	Y =   -630.910  mm,	Z =   -257.219  mm,
	W =  90.000 deg,	P =   0.000 deg,	R =   90.000 deg
};
P[2057]{
   GP1:
	UF : 0, UT : 6,		CONFIG : 'N U T, 0, 0, 0',
	X =  32.561  mm,	Y =   -631.845  mm,	Z =   -257.299  mm,
	W =  90.000 deg,	P =   0.000 deg,	R =   90.000 deg
};
P[2058]{
   GP1:
	UF : 0, UT : 6,		CONFIG : 'N U T, 0, 0, 0',
	X =  37.129  mm,	Y =   -639.988  mm,	Z =   -256.975  mm,
	W =  90.000 deg,	P =   0.000 deg,	R =   90.000 deg
};
P[2059]{
   GP1:
	UF : 0, UT : 6,		CONFIG : 'N U T, 0, 0, 0',
	X =  38.031  mm,	Y =   -641.453  mm,	Z =   -257.113  mm,
	W =  90.000 deg,	P =   0.000 deg,	R =   90.000 deg
};
P[2060]{
   GP1:
	UF : 0, UT : 6,		CONFIG : 'N U T, 0, 0, 0',
	X =  38.433  mm,	Y =   -642.006  mm,	Z =   -257.313  mm,
	W =  90.000 deg,	P =   0.000 deg,	R =   90.000 deg
};
P[2061]{
   GP1:
	UF : 0, UT : 6,		CONFIG : 'N U T, 0, 0, 0',
	X =  39.005  mm,	Y =   -642.978  mm,	Z =   -257.340  mm,
	W =  90.000 deg,	P =   0.000 deg,	R =   90.000 deg
};
P[2062]{
   GP1:
	UF : 0, UT : 6,		CONFIG : 'N U T, 0, 0, 0',
	X =  39.311  mm,	Y =   -643.617  mm,	Z =   -257.186  mm,
	W =  90.000 deg,	P =   0.000 deg,	R =   90.000 deg
};
P[2063]{
   GP1:
	UF : 0, UT : 6,		CONFIG : 'N U T, 0, 0, 0',
	X =  40.799  mm,	Y =   -646.278  mm,	Z =   -257.069  mm,
	W =  90.000 deg,	P =   0.000 deg,	R =   90.000 deg
};
P[2064]{
   GP1:
	UF : 0, UT : 6,		CONFIG : 'N U T, 0, 0, 0',
	X =  42.323  mm,	Y =   -648.806  mm,	Z =   -257.226  mm,
	W =  90.000 deg,	P =   0.000 deg,	R =   90.000 deg
};
P[2065]{
   GP1:
	UF : 0, UT : 6,		CONFIG : 'N U T, 0, 0, 0',
	X =  43.261  mm,	Y =   -650.424  mm,	Z =   -257.235  mm,
	W =  90.000 deg,	P =   0.000 deg,	R =   90.000 deg
};
P[2066]{
   GP1:
	UF : 0, UT : 6,		CONFIG : 'N U T, 0, 0, 0',
	X =  46.573  mm,	Y =   -656.087  mm,	Z =   -257.338  mm,
	W =  90.000 deg,	P =   0.000 deg,	R =   90.000 deg
};
P[2067]{
   GP1:
	UF : 0, UT : 6,		CONFIG : 'N U T, 0, 0, 0',
	X =  48.251  mm,	Y =   -659.098  mm,	Z =   -257.189  mm,
	W =  90.000 deg,	P =   0.000 deg,	R =   90.000 deg
};
P[2068]{
   GP1:
	UF : 0, UT : 6,		CONFIG : 'N U T, 0, 0, 0',
	X =  50.434  mm,	Y =   -662.894  mm,	Z =   -257.167  mm,
	W =  90.000 deg,	P =   0.000 deg,	R =   90.000 deg
};
P[2069]{
   GP1:
	UF : 0, UT : 6,		CONFIG : 'N U T, 0, 0, 0',
	X =  51.268  mm,	Y =   -664.147  mm,	Z =   -257.277  mm,
	W =  90.000 deg,	P =   0.000 deg,	R =   90.000 deg
};
P[2070]{
   GP1:
	UF : 0, UT : 6,		CONFIG : 'N U T, 0, 0, 0',
	X =  51.615  mm,	Y =   -664.653  mm,	Z =   -257.253  mm,
	W =  90.000 deg,	P =   0.000 deg,	R =   90.000 deg
};
P[2071]{
   GP1:
	UF : 0, UT : 6,		CONFIG : 'N U T, 0, 0, 0',
	X =  52.878  mm,	Y =   -666.299  mm,	Z =   -257.243  mm,
	W =  90.000 deg,	P =   0.000 deg,	R =   90.000 deg
};
P[2072]{
   GP1:
	UF : 0, UT : 6,		CONFIG : 'N U T, 0, 0, 0',
	X =  54.141  mm,	Y =   -667.440  mm,	Z =   -257.302  mm,
	W =  90.000 deg,	P =   0.000 deg,	R =   90.000 deg
};
P[2073]{
   GP1:
	UF : 0, UT : 6,		CONFIG : 'N U T, 0, 0, 0',
	X =  54.757  mm,	Y =   -668.129  mm,	Z =   -257.058  mm,
	W =  90.000 deg,	P =   0.000 deg,	R =   90.000 deg
};
P[2074]{
   GP1:
	UF : 0, UT : 6,		CONFIG : 'N U T, 0, 0, 0',
	X =  55.555  mm,	Y =   -668.641  mm,	Z =   -257.050  mm,
	W =  90.000 deg,	P =   0.000 deg,	R =   90.000 deg
};
P[2075]{
   GP1:
	UF : 0, UT : 6,		CONFIG : 'N U T, 0, 0, 0',
	X =  57.095  mm,	Y =   -669.383  mm,	Z =   -257.283  mm,
	W =  90.000 deg,	P =   0.000 deg,	R =   90.000 deg
};
P[2076]{
   GP1:
	UF : 0, UT : 6,		CONFIG : 'N U T, 0, 0, 0',
	X =  58.715  mm,	Y =   -670.086  mm,	Z =   -257.143  mm,
	W =  90.000 deg,	P =   0.000 deg,	R =   90.000 deg
};
P[2077]{
   GP1:
	UF : 0, UT : 6,		CONFIG : 'N U T, 0, 0, 0',
	X =  59.374  mm,	Y =   -670.169  mm,	Z =   -257.322  mm,
	W =  90.000 deg,	P =   0.000 deg,	R =   90.000 deg
};
P[2078]{
   GP1:
	UF : 0, UT : 6,		CONFIG : 'N U T, 0, 0, 0',
	X =  62.959  mm,	Y =   -670.580  mm,	Z =   -257.346  mm,
	W =  90.000 deg,	P =   0.000 deg,	R =   90.000 deg
};
P[2079]{
   GP1:
	UF : 0, UT : 6,		CONFIG : 'N U T, 0, 0, 0',
	X =  69.236  mm,	Y =   -669.008  mm,	Z =   -257.165  mm,
	W =  90.000 deg,	P =   0.000 deg,	R =   90.000 deg
};
P[2080]{
   GP1:
	UF : 0, UT : 6,		CONFIG : 'N U T, 0, 0, 0',
	X =  71.953  mm,	Y =   -667.428  mm,	Z =   -257.346  mm,
	W =  90.000 deg,	P =   0.000 deg,	R =   90.000 deg
};
P[2081]{
   GP1:
	UF : 0, UT : 6,		CONFIG : 'N U T, 0, 0, 0',
	X =  75.997  mm,	Y =   -665.098  mm,	Z =   -257.336  mm,
	W =  90.000 deg,	P =   0.000 deg,	R =   90.000 deg
};
P[2082]{
   GP1:
	UF : 0, UT : 6,		CONFIG : 'N U T, 0, 0, 0',
	X =  76.889  mm,	Y =   -664.572  mm,	Z =   -257.362  mm,
	W =  90.000 deg,	P =   0.000 deg,	R =   90.000 deg
};
P[2083]{
   GP1:
	UF : 0, UT : 6,		CONFIG : 'N U T, 0, 0, 0',
	X =  78.628  mm,	Y =   -663.590  mm,	Z =   -257.310  mm,
	W =  90.000 deg,	P =   0.000 deg,	R =   90.000 deg
};
P[2084]{
   GP1:
	UF : 0, UT : 6,		CONFIG : 'N U T, 0, 0, 0',
	X =  80.682  mm,	Y =   -662.518  mm,	Z =   -257.033  mm,
	W =  90.000 deg,	P =   0.000 deg,	R =   90.000 deg
};
P[2085]{
   GP1:
	UF : 0, UT : 6,		CONFIG : 'N U T, 0, 0, 0',
	X =  87.768  mm,	Y =   -658.486  mm,	Z =   -256.890  mm,
	W =  90.000 deg,	P =   0.000 deg,	R =   90.000 deg
};
P[2086]{
   GP1:
	UF : 0, UT : 6,		CONFIG : 'N U T, 0, 0, 0',
	X =  88.444  mm,	Y =   -657.992  mm,	Z =   -257.140  mm,
	W =  90.000 deg,	P =   0.000 deg,	R =   90.000 deg
};
P[2087]{
   GP1:
	UF : 0, UT : 6,		CONFIG : 'N U T, 0, 0, 0',
	X =  89.560  mm,	Y =   -657.300  mm,	Z =   -257.256  mm,
	W =  90.000 deg,	P =   0.000 deg,	R =   90.000 deg
};
P[2088]{
   GP1:
	UF : 0, UT : 6,		CONFIG : 'N U T, 0, 0, 0',
	X =  90.813  mm,	Y =   -656.656  mm,	Z =   -257.064  mm,
	W =  90.000 deg,	P =   0.000 deg,	R =   90.000 deg
};
P[2089]{
   GP1:
	UF : 0, UT : 6,		CONFIG : 'N U T, 0, 0, 0',
	X =  92.316  mm,	Y =   -655.716  mm,	Z =   -257.239  mm,
	W =  90.000 deg,	P =   0.000 deg,	R =   90.000 deg
};
P[2090]{
   GP1:
	UF : 0, UT : 6,		CONFIG : 'N U T, 0, 0, 0',
	X =  93.337  mm,	Y =   -655.185  mm,	Z =   -257.097  mm,
	W =  90.000 deg,	P =   0.000 deg,	R =   90.000 deg
};
P[2091]{
   GP1:
	UF : 0, UT : 6,		CONFIG : 'N U T, 0, 0, 0',
	X =  96.339  mm,	Y =   -653.441  mm,	Z =   -257.122  mm,
	W =  90.000 deg,	P =   0.000 deg,	R =   90.000 deg
};
P[2092]{
   GP1:
	UF : 0, UT : 6,		CONFIG : 'N U T, 0, 0, 0',
	X =  97.336  mm,	Y =   -652.870  mm,	Z =   -257.110  mm,
	W =  90.000 deg,	P =   0.000 deg,	R =   90.000 deg
};
P[2093]{
   GP1:
	UF : 0, UT : 6,		CONFIG : 'N U T, 0, 0, 0',
	X =  97.896  mm,	Y =   -652.463  mm,	Z =   -257.311  mm,
	W =  90.000 deg,	P =   0.000 deg,	R =   90.000 deg
};
P[2094]{
   GP1:
	UF : 0, UT : 6,		CONFIG : 'N U T, 0, 0, 0',
	X =  101.660  mm,	Y =   -650.342  mm,	Z =   -257.185  mm,
	W =  90.000 deg,	P =   0.000 deg,	R =   90.000 deg
};
P[2095]{
   GP1:
	UF : 0, UT : 6,		CONFIG : 'N U T, 0, 0, 0',
	X =  106.888  mm,	Y =   -647.256  mm,	Z =   -257.349  mm,
	W =  90.000 deg,	P =   0.000 deg,	R =   90.000 deg
};
P[2096]{
   GP1:
	UF : 0, UT : 6,		CONFIG : 'N U T, 0, 0, 0',
	X =  111.389  mm,	Y =   -644.778  mm,	Z =   -257.059  mm,
	W =  90.000 deg,	P =   0.000 deg,	R =   90.000 deg
};
P[2097]{
   GP1:
	UF : 0, UT : 6,		CONFIG : 'N U T, 0, 0, 0',
